	aAMSNetID	AT %I* 	:	AMSNETID;
	wSlaveADDR	AT %I*			:	WORD;
	PLCResetRequired	:	BOOL := FALSE;		
END_VAR

VAR_INPUT
	b_EnablePower 			: BOOL;
	r_CoolantTemperature 	: REAL;
END_VAR

VAR_OUTPUT
	Get : ST_HeatpumpSystemGet;
END_VAR

VAR
	PrimaryHeatpump_EnablePower		AT %Q* :	BOOL;
	SecondaryHeatpump_EnablePower	AT %Q* :	BOOL;
	b_AuxilliaryHeaterEnable		AT %Q*	:	Bool;
END_VAR

UpdateRTUSettings();				

CASE st_params.HeatpumpType OF
	eSupportedHeatpumps.TranePicco:
		PrimaryHeatpump := TraneHeatpump[0];
		TraneHeatpump[0](MBMaster := MBMaster, 
			ACPowerStatus := b_EnablePower,  
			st_params := st_params, 
			HeatPumpId := st_Params.PrimaryHeatpumpAddr);
		get.PrimaryHeatpumpGet REF= TraneHeatpump[0].Get;
				
	eSupportedHeatpumps.LgThermaV:
		PrimaryHeatpump := LGHeatpump[0];
		LGHeatpump[0](MBMaster := MBMaster, 
			ACPowerStatus := b_EnablePower,  
			st_params := st_params, 
			HeatPumpId := st_Params.PrimaryHeatpumpAddr);
		get.PrimaryHeatpumpGet REF= lgHeatpump[0].Get;
END_CASE

get.SecondaryHeatpumpGet REF= lgHeatpump[1].Get;

IF ST_Params.b_DoubleHeatpump THEN
	CASE st_params.HeatpumpType OF
		eSupportedHeatpumps.TranePicco:		
			SecondaryHeatpump := TraneHeatpump[1];
			TraneHeatpump[1](MBMaster := MBMaster, 
				ACPowerStatus := b_EnablePower,  
				st_params := st_params, 
				HeatPumpId := st_Params.SecondaryHeatpumpAddr,
				get => get.SecondaryHeatpumpGet);
		eSupportedHeatpumps.LgThermaV:		
			SecondaryHeatpump := LGHeatpump[1];	
			LGHeatpump[1](MBMaster := MBMaster, 
				ACPowerStatus := b_EnablePower,  
				st_params := st_params, 
				HeatPumpId := st_Params.SecondaryHeatpumpAddr,
				get => get.SecondaryHeatpumpGet);
	END_CASE
END_IF

get.HeatPumpStatus := get.PrimaryHeatpumpGet.HeatPumpState;
get.PrimaryHeatpumpGet.HeatpumpData.r_CoolantPower := CalculateCoolantPower();

PowerControl();
setMBControl();

METHOD CalculateCoolantPower : REAL
VAR_INST
	PowerMA : fb_MovingAverage := (enable := TRUE);
	ActualPower : REAL;
	
	deltaT :  REAL;
	cp	: REAL;
	Flow : REAL;
	
	ton_synctimer	: TON := (PT:= T#1S);
END_VAR
flow	:= get.PrimaryHeatpumpGet.HeatpumpData.ui_WaterFlowRate;
deltaT	:= get.PrimaryHeatpumpGet.HeatpumpData.r_InletWaterTemp - get.PrimaryHeatpumpGet.HeatpumpData.r_OutletWaterTemp;
cp		:= 3.647;

ton_synctimer(IN := NOT ton_synctimer.Q);

ActualPower := (flow * cp * deltaT * 1.05) / 0.06;

IF ton_synctimer.Q THEN
	PowerMA(IN := ActualPower, length:= 15);
END_IF

CalculateCoolantPower := PowerMA.Q;
END_METHOD

METHOD EMStop : BOOL
VAR_INPUT
END_VAR
EMstop := PrimaryHeatpump.emstop() and SecondaryHeatpump.emstop();
END_METHOD

METHOD GetDiagnostics 
VAR_IN_OUT
	AddError		: ARRAY [*] OF FB_AddErrorST;
	a_ActiveEvents	: ARRAY [*] OF ST_ErrorStruct;
	w_Index			: WORD;
END_VAR

VAR_OUTPUT
	b_errorActive	: BOOL;
	b_warningActive	: BOOL;
END_VAR

VAR
	by_errCt	: BYTE;
	by_warnCt	: BYTE;
	w_ID		: WORD;
END_VAR
(*Heatpump Heating inhibited*)	AddError[w_Index](
			b_ErrorTrig				:= b_AuxilliaryHeaterEnable,
			out_ST_Error			:= a_ActiveEvents[w_Index],
			w_ErrorID				:= 20,
			s_Message				:= 'Coolant undertemperature error, heatpump heating inhibited',
			e_sev					:= eSeverity.Info,	
			b_AutoClear				:= TRUE,
			);
		w_Index := w_Index +1;	
		
(*Heatpump type changed*)	AddError[w_Index](
			b_ErrorTrig				:= PLCResetRequired,
			out_ST_Error			:= a_ActiveEvents[w_Index],
			w_ErrorID				:= 21,
			s_Message				:= 'Heatpump type changed, Reset PLC to activate new settings',
			e_sev					:= eSeverity.Warning,	
			b_AutoClear				:= TRUE,
			);
		w_Index := w_Index +1;	

(*Heatpump type changed*)	AddError[w_Index](
			b_ErrorTrig				:= PLCResetRequired,
			out_ST_Error			:= a_ActiveEvents[w_Index],
			w_ErrorID				:= 22,
			s_Message				:= 'Heatpump not operational until PLC has been restarted!',
			e_sev					:= eSeverity.Warning,	
			b_AutoClear				:= TRUE,
			);
		w_Index := w_Index +1;	

//check if this call works:
PrimaryHeatpump.GetDiagnostics(AddError := AddError, a_ActiveEvents := a_ActiveEvents, w_Index := w_Index, b_errorActive => b_errorActive, b_warningActive => b_warningActive);
SecondaryHeatpump.GetDiagnostics(AddError := AddError, a_ActiveEvents := a_ActiveEvents, w_Index := w_Index, b_errorActive => b_errorActive, b_warningActive => b_warningActive);
END_METHOD

METHOD GetWearCounters : BOOL
VAR_INST
	MstrPowerCycles				:	FB_Varlogger;
	MstrPowerHours				:	FB_Varlogger;
	
	MstrCompressorCycles		:	FB_Varlogger;
	MstrWaterpumpHours			:	FB_Varlogger;
	
	SlowDataTimer				:	TON := (PT := T#1H);
END_VAR
SlowDataTimer(IN := NOT SlowDataTimer.Q);

MstrPowerCycles(		TriggerInput := PrimaryHeatpump_EnablePower,
						LogItemGroup := eLogItemGroupID.CoolingSystem, 
						LogItemName := 'MstrHPPwrCnt', 
						LogType := eLogtypes.TrackCycles);
						
MstrPowerCycles(		TriggerInput := PrimaryHeatpump_EnablePower,
						LogItemGroup := eLogItemGroupID.CoolingSystem, 
						LogItemName := 'MstrHPPwrHrs', 
						LogType := eLogtypes.TrackOnTime);

IF get.PrimaryHeatpumpGet.HeatpumpData.i_OperatingHours > 0 THEN
	Wearlogging.SetInteger(eLogItemGroupID.CoolingSystem, 	'MstrHPCompHrs', 			eLogTypes.WriteValue, 		INT_TO_LINT(get.PrimaryHeatpumpGet.HeatpumpData.i_OperatingHours));
END_IF

MstrCompressorCycles(	TriggerInput := ((get.PrimaryHeatpumpGet.HeatpumpData.r_HighPressure-get.PrimaryHeatpumpGet.HeatpumpData.r_LowPressure)>5), //test this
						LogItemGroup :=  eLogItemGroupID.CoolingSystem, 
						LogItemName := 'MstrHPCompCnt', 
						LogType := eLogtypes.TrackCycles);
END_METHOD

METHOD PRIVATE PowerControl : BOOL
VAR_INST
	PowerOnDelay1: TON := (PT := TIME#1S);
	PowerOnDelay2: TON := (PT := TIME#2S);
END_VAR

//heatpump 2 is enabled with a delay to limit inrush
PowerOnDelay1(in:= b_EnablePower, Q=>PrimaryHeatpump_EnablePower);
PowerOnDelay2(IN := b_EnablePower AND st_params.b_DoubleHeatpump ,Q=> SecondaryHeatpump_EnablePower);
END_METHOD

METHOD Reset : BOOL
VAR_INPUT
END_VAR
Reset := PrimaryHeatpump.Reset() and SecondaryHeatpump.Reset();
END_METHOD

METHOD PRIVATE SetMBControl : BOOL
VAR_INST
	ton_MaximumMBTimeframe	:	TON := (PT := TIME#10S);

	CommFreeForID			: BYTE := 0;
	CommFreeTimeout			: TON := (PT := TIME#10S);	
END_VAR
//500ms trigger to switch MB bus ownership to next heatpump
ton_MaximumMBTimeframe(in := NOT ton_MaximumMBTimeframe.Q);

IF NOT PrimaryHeatpump.MBCommBusy() AND NOT SecondaryHeatpump.MBCommBusy() THEN
	CommFreeForID := (CommFreeForID+1);
END_IF
	
PrimaryHeatPump.AllowMBComm(b_AllowComm := (CommFreeForID=1));
SecondaryHeatPump.AllowMBComm(b_AllowComm := (CommFreeForID=2));

IF CommFreeForID > SEL(st_params.b_DoubleHeatpump, 1, 2) THEN
	CommFreeForID := 0;
END_IF
END_METHOD

METHOD Shutdown : BOOL
VAR_INPUT
END_VAR
HeatPumpOperationAllowed := FALSE;
END_METHOD

METHOD Start : BOOL
VAR_INPUT
END_VAR
HeatpumpOperationAllowed := true;
END_METHOD

METHOD UpdateRTUSettings : BOOL
VAR_INPUT
END_VAR

VAR_INST
	CurrentBussettings			:	WORD 	:=  0;
	MethodSTate					:	UINT	:=	0;
	CoEWrite					:	FB_EcCoeSdoWriteEx;
	CoERead						:	FB_EcCoeSdoReadEx;
	Netid						:	T_AMSNETID;
	
	Testoutput					:	UDINT;
	Testbool					:	BOOL;
	TestBool2					:	BOOL;
	CurrentBusSetting			:   WORD;	
	RequiredBusSetting			:	WORD;	
	COEReadDone					:	F_trig;
	COEWriteDone				:	F_trig;
END_VAR
Netid := F_CreateAmsNetId(aAMSNetID);

CoERead(sNetID := Netid,
		nSlaveAddr := wSlaveADDR,
		nSubIndex := 0,
		nIndex := 16#4074,
		pDstBuf := ADR(CurrentBusSetting),
		cbBufLen := SIZEOF(CurrentBusSetting),
		tTimeout := T#1S,
		bCompleteAccess := TRUE,
		cbRead => Testoutput);

CoEWrite(sNetID := Netid,
		nSlaveAddr := wSlaveADDR,
		nSubIndex := 0,
		nIndex := 16#4074,
		pSRCBuf := ADR(RequiredBusSetting),
		cbBufLen := SIZEOF(RequiredBusSetting),
		tTimeout := T#1S,
		bCompleteAccess := TRUE);

COEReadDone(clk:= CoERead.bBusy);
COEwriteDone(clk:= CoEWrite.bBusy);


CASE MethodSTate OF
	0:	//init
		CoERead(bExecute := FALSE);
		CoEwrite(bExecute := FALSE);
		MethodSTate := 1;
	1:	//ReadCurrentSettings
		CoERead(bExecute := TRUE);
		IF COEReadDone.q THEN
			IF NOT CoERead.bError THEN
				MethodSTate := 2;
			END_IF
			CoERead(bExecute := FALSE);
		END_IF
	2:	//idle
		IF (st_params.HeatpumpType = eSupportedHeatpumps.LgThermaV AND CurrentBusSetting <> 3) THEN
			RequiredBusSetting := 3;
			MethodSTate := 3; //write new settings
		ELSIF(st_params.HeatpumpType = eSupportedHeatpumps.TranePicco AND CurrentBusSetting <> 4) THEN
			RequiredBusSetting := 4;			
			MethodSTate := 3; //write new settings
		END_IF
	3: //write new settings
		CoEwrite(bExecute := TRUE);
		IF COEWriteDone.q THEN
			CoEwrite(bExecute := False);
			IF NOT CoERead.bError THEN
				MethodSTate := 4;
			END_IF
			CoERead(bExecute := FALSE);
		END_IF
	4:	//Wait for reboot to activate settings
			PLCResetRequired := TRUE;
		
END_CASE
END_METHOD

METHOD WriteSetpoint : BOOL
VAR_INPUT
	OperatingMode	:	eHeatpumpMode := eHeatpumpMode.Standby;
	SetPoint		: 	REAL := 18.0;
END_VAR
IF HeatpumpOperationAllowed THEN
	IF Operatingmode = eHeatpumpMode.Heating AND r_CoolantTemperature < st_params.r_MinimumCoolantTemperatureForHPHeatingMode THEN
		PrimaryHeatpump.Setpoint(eHeatpumpMode.Standby, Temperature := 18.0);
		b_AuxilliaryHeaterEnable := TRUE;
	ELSE
		PrimaryHeatpump.Setpoint(OperatingMode := OperatingMode, Temperature:=SetPoint);
		b_AuxilliaryHeaterEnable := FALSE;
	END_IF
ELSE
	PrimaryHeatpump.Setpoint(eHeatpumpMode.Standby, Temperature := 18.0);
	b_AuxilliaryHeaterEnable := FALSE;
END_IF
//This method will also contain potential master/slave temperature differentials and other differences between heatpumps
//Heatpumps[2].WriteSetpoint(OperatingMode := OperatingMode);
END_METHOD

END_FUNCTION_BLOCK

// ---- POUs/Objects/CoolingSystem/HeatpumpSystem/FB_LGHeatpump.TcPOU
FUNCTION_BLOCK FB_LGHeatpump implements IF_Heatpump
VAR_IN_OUT
	MBMaster		:	ModbusRtuMasterV2_KL6x22B;
END_VAR

VAR_OUTPUT
	Get				:	ST_HeatPump_Get;

END_VAR

VAR_IN_OUT CONSTANT
	st_params		: 	ST_Coolingsystem_params;
END_VAR

VAR_INPUT
	ACPowerStatus	:	BOOL;
	HeatPumpID		:	BYTE;
	SFCInit			:	BOOL;
	e_ID				:	eObject_ID := eObject_ID.HeatPump;
END_VAR
		
VAR
	ton_MBBUSYTimeOut		: TON := (PT := T#10s);
	DataBuffer				:	ARRAY[0..50] OF WORD;
	ton_modbusStuckTrigger	:	Ton	:=	(PT := T#5S);
	Ton_ErrorTimer			:	Ton := (PT := T#5M);
	MBRetryCount			:	BYTE;
	MBFree					:	BOOL;
	bMBActive				:	BOOL;
	ftrig_ModbusStartTrigger		:	f_Trig;
	TransmissionDoneTrigger	:	F_Trig;
	rtrig_ManualModbusStartTrigger : r_trig;
	btest	:	BOOL;
	ManADDR : BYTE;
	ton_testTimer	:	Ton := (Pt := T#100MS);
	TP_ModbusStartTriggerDelay	:	TP := (PT := TIME#50MS);
	u_counter				:	UINT;
END_VAR

VAR
	RequestedSetpoint				:	st_OperatingPoint;
	b_EMStop						:	BOOL;
	b_resetErrors					:	BOOL;
	t_RemainingPreheatingTime	:	TIME;
	sPressureErrorText			:	STRING;
	sCompressorErrorText		:	STRING;
	sPumpErrorText				:	STRING;
	sWaterTempErrorText			:	STRING;
END_VAR

VAR PERSISTENT
	dt_LastHPOperationTime	:	DT := DT#1970-1-1-0:0:0.000;
END_VAR


VAR
	CoilStatus		:	BYTE;
	LGget	:	LG_get;
	LGset	:	LG_SET;

	HeatpumpEMOperationAvailable	:	Bool;
END_VAR

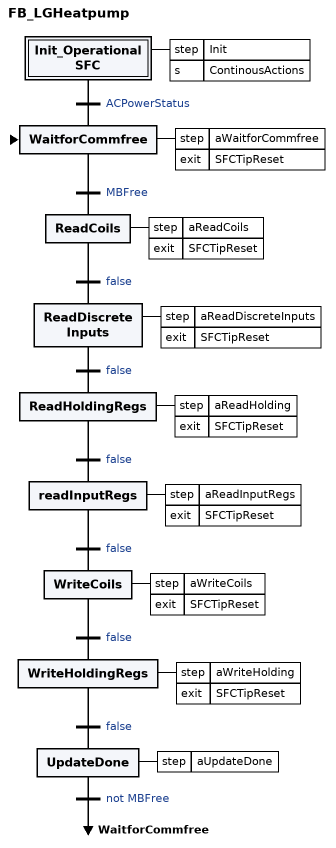
INITIAL_STEP Init_OperationalSFC:
    Init(N);  // step action
    ContinousActions(s);
END_STEP
TRANSITION FROM Init_OperationalSFC TO WaitforCommfree
    := ACPowerStatus;
END_TRANSITION
STEP WaitforCommfree:
    aWaitforCommfree(N);  // step action
    SFCTipReset(P0);  // exit action
END_STEP
TRANSITION FROM WaitforCommfree TO ReadCoils
    := MBFree;
END_TRANSITION
STEP ReadCoils:  // max time T#2S
    aReadCoils(N);  // step action
    SFCTipReset(P0);  // exit action
END_STEP
TRANSITION FROM ReadCoils TO ReadDiscreteInputs
    := false;
END_TRANSITION
STEP ReadDiscreteInputs:
    aReadDiscreteInputs(N);  // step action
    SFCTipReset(P0);  // exit action
END_STEP
TRANSITION FROM ReadDiscreteInputs TO ReadHoldingRegs
    := false;
END_TRANSITION
STEP ReadHoldingRegs:
    aReadHolding(N);  // step action
    SFCTipReset(P0);  // exit action
END_STEP
TRANSITION FROM ReadHoldingRegs TO readInputRegs
    := false;
END_TRANSITION
STEP readInputRegs:
    aReadInputRegs(N);  // step action
    SFCTipReset(P0);  // exit action
END_STEP
TRANSITION FROM readInputRegs TO WriteCoils
    := false;
END_TRANSITION
STEP WriteCoils:
    aWriteCoils(N);  // step action
    SFCTipReset(P0);  // exit action
END_STEP
TRANSITION FROM WriteCoils TO WriteHoldingRegs
    := false;
END_TRANSITION
STEP WriteHoldingRegs:
    aWriteHolding(N);  // step action
    SFCTipReset(P0);  // exit action
END_STEP
TRANSITION FROM WriteHoldingRegs TO UpdateDone
    := false;
END_TRANSITION
STEP UpdateDone:
    aUpdateDone(N);  // step action
END_STEP
TRANSITION FROM UpdateDone TO WaitforCommfree
    := not MBFree;
END_TRANSITION

METHOD AllowMBComm : BOOL
VAR_INPUT
	b_AllowComm	:	Bool;
END_VAR
MBFree	:= b_AllowComm;
END_METHOD

ACTION aReadCoils:
bMBActive := TRUE;

MBMaster.ReadCoils(	UnitID 		:= 	HeatPumpID,
					Quantity 	:= 	5,
					MBAddr		:=	0,				
					cbLength 	:= 	6,
					pMemoryAddr	:=	ADR(CoilStatus),
					Execute		:=	ftrig_ModbusStartTrigger.Q,
				);
	

IF TransmissionDoneTrigger.q THEN
	IF NOT MBMaster.Error THEN
		//Full datastruct for debug purposes. Can be removed later
		LGget.Coils.b_EnableOperation := CoilStatus.0;
		LGget.Coils.b_EnableSwwOperation := CoilStatus.1;
		LGget.Coils.b_EnableSilentMode := CoilStatus.2;
		LGget.Coils.b_EnableDesinfectionMode := Coilstatus.3;
		LGget.Coils.b_EmstopActive := CoilStatus.4;
		LGget.Coils.b_EnableEmStop := CoilStatus.5;
		//Full datastruct for debug purposes. Can be removed later
		
	ELSE
		MBRetryCount := MBRetryCount + 1;
	END_IF
	
	sfctip := TRUE;
END_IF


get.HeatpumpData.w_ErrorList[1] := lgget.Data.UI_ErrorCode;
get.Setpoint := lgget.Control.r_Setpoint1;
END_ACTION

ACTION aReadDiscreteInputs:


MBMaster.ReadInputStatus(	UnitID 		:= 	HeatPumpID,
							Quantity 	:= 	16,
							MBAddr		:=	0,
							cbLength 	:= 	SIZEOF(Databuffer),
							pMemoryAddr	:=	ADR(DataBuffer),
							Execute		:=	ftrig_ModbusStartTrigger.Q,
						);



IF TransmissionDoneTrigger.q THEN
	IF NOT MBMaster.Error THEN
		//Full datastruct for debug purposes. Can be removed later
		LGget.Status.b_WaterFlowNOK := DataBuffer[0].0;
		LGget.Status.b_WaterPumpOn := DataBuffer[0].1;
		LGget.Status.b_ExtWaterPumpOn := DataBuffer[0].2;
		LGget.Status.b_CompressorOn := DataBuffer[0].3;
		LGget.Status.b_DefrostOn := DataBuffer[0].4;
		LGget.Status.b_SWWModeOn := DataBuffer[0].5;
		LGget.Status.b_SWWTankDesinfectionActive := DataBuffer[0].6;
		LGget.Status.b_SilentModeOn := DataBuffer[0].7;
		LGget.Status.b_CoolingActive := DataBuffer[0].8;
		LGget.Status.b_SolarPumpActive := DataBuffer[0].9;
		LGget.Status.b_BackupHeater1Active := DataBuffer[0].10;
		LGget.Status.b_BackupHeater2Active := DataBuffer[0].11;
		LGget.Status.b_SWWBoostHeaterActive := DataBuffer[0].12;
		LGget.Status.b_ErrorActive := DataBuffer[0].13;
		LGget.Status.b_EMOperationAvailable := DataBuffer[0].14;
		LGget.Status.b_EMSWWOperationAvailable := DataBuffer[0].15;
		LGget.Status.b_MixPumpActive := DataBuffer[1].0;
		//Full datastruct for debug purposes. Can be removed later
		
		get.Events.b_PumpError := DataBuffer[0].0;
		get.HeatpumpData.b_DefrostingActive := DataBuffer[0].4;
		
		
		//error active and no em operation allowed
		IF DataBuffer[0].13 THEN
			get.HeatPumpState := eHeatpumpstate.ERROR;
			IF NOT DataBuffer[0].14 THEN
				HeatpumpEMOperationAvailable := FALSE;
			ELSE
				HeatpumpEMOperationAvailable := TRUE;
			END_IF
		ELSIF get.HeatPumpState = eHeatpumpstate.ERROR THEN
			get.HeatPumpState := eHeatpumpstate.Initializing;
			HeatpumpEMOperationAvailable := FALSE;
		END_IF
		
		//done, preset for next step
		MBRetryCount := 0;
	ELSE
		MBRetryCount := MBRetryCount + 1;
	END_IF
	sfctip := TRUE;
END_IF
END_ACTION

ACTION aReadHolding:

MBMaster.ReadRegs(	UnitID 		:= 	HeatPumpID,
					Quantity 	:= 	10,
					MBAddr		:=	0,
					cbLength 	:= 	SIZEOF(Databuffer),
					pMemoryAddr	:=	ADR(DataBuffer),
					Execute		:=	ftrig_ModbusStartTrigger.Q,
					);


IF TransmissionDoneTrigger.q THEN
	IF NOT MBMaster.Error THEN
		LGget.Control.ui_OperatingMode := Databuffer[0];
		LGget.Control.ui_ControlMode := Databuffer[1];
		LGget.Control.r_Setpoint1 := (WORD_TO_REAL(Databuffer[2])/10);
		LGget.Control.r_RoomSetpoint := (WORD_TO_REAL(Databuffer[3])/10);
		LGget.Control.ui_TempShiftValue := Databuffer[4];
		LGget.Control.r_Setpoint2 := (WORD_TO_REAL(Databuffer[5])/10);
		LGget.Control.r_RoomSetpoint2 := (WORD_TO_REAL(Databuffer[6])/10);
		LGget.Control.ui_TempShiftValue2 := Databuffer[7];
		LGget.Control.r_DHWgoalTemp := (WORD_TO_REAL(Databuffer[8])/10);
		LGget.Control.ui_EnergyStatus := Databuffer[9];
		
		get.Setpoint := (WORD_TO_REAL(Databuffer[2])/10);


		IF get.HeatPumpState <> eHeatpumpstate.ERROR THEN
			CASE lgget.Data.ui_OperationalMode OF
				0:
					get.HeatPumpState := eHeatpumpstate.Standby;
				1:
					get.HeatPumpState := eHeatpumpstate.Active_Cooling;
				2:
					get.HeatPumpState := eHeatpumpstate.Active_Heating;
			END_CASE
		END_IF
	
		//done, preset for next step
		MBRetryCount := 0;

	ELSE
		MBRetryCount := MBRetryCount + 1;
		
	END_IF
	sfctip := TRUE;
END_IF
END_ACTION

ACTION aReadInputRegs:
//SFCTip := FALSE;

MBMaster.ReadInputRegs ( 
					UnitID 		:= 	HeatPumpID,
					Quantity 	:= 	13,
					MBAddr		:=	0,
					cbLength 	:= 	SIZEOF(Databuffer),
					pMemoryAddr	:=	ADR(Databuffer),
					Execute		:=	ftrig_ModbusStartTrigger.Q,		
					);
				
IF TransmissionDoneTrigger.q THEN
	IF NOT MBMaster.Error THEN
		
	//Full datastruct for debug purposes. Can be removed later
		LGget.Data.UI_ErrorCode := Databuffer[0];	
		LGget.Data.ui_OperationalMode := (Databuffer[1]);	
		LGget.Data.r_CoolantInletTemp := WORD_TO_REAL((Databuffer[2]))/10;	
		LGget.Data.r_CoolantOutletTemp := WORD_TO_REAL((Databuffer[3]))/10;
		LGget.Data.r_BackupHeaterTemp := WORD_TO_REAL((Databuffer[4]))/10;
		LGget.Data.r_SWWTankTemp :=  WORD_TO_REAL((Databuffer[5]))/10;
		LGget.Data.r_SolarCollectorTemp := WORD_TO_REAL((Databuffer[6]))/10;
		LGget.Data.r_RoomTemp1 := WORD_TO_REAL((Databuffer[7]))/10;
		LGget.Data.r_FlowRate := WORD_TO_REAL((Databuffer[8]))/10;
		LGget.Data.r_FlowTempCircuit2 := WORD_TO_REAL((Databuffer[9]))/10;
		LGget.Data.r_RoomTemp2 := WORD_TO_REAL((Databuffer[10]))/10;
		LGget.Data.UI_EnergyStatus := (Databuffer[11]);
		LGget.Data.r_OutsideTemp := WORD_TO_REAL((Databuffer[12]))/10;
	//full datastruct for debug purposes. can be removed later	
		
		
		get.HeatpumpData.w_ErrorList[1] := Databuffer[0];
		Get.HeatpumpData.r_InletWaterTemp := WORD_TO_REAL((Databuffer[2]))/10;	
		get.HeatpumpData.r_OutletWaterTemp := WORD_TO_REAL((Databuffer[3]))/10;
		get.HeatpumpData.r_OutdoorTemp := WORD_TO_REAL((Databuffer[12]))/10;
		get.HeatpumpData.ui_WaterFlowRate := TO_UINT(Databuffer[8]/10);
	ELSE
		MBRetryCount := MBRetryCount + 1;
	END_IF
	sfctip := TRUE;
END_IF
END_ACTION

ACTION aUpdateDone:
SFCTip := FALSE;
bMBActive := FALSE;
END_ACTION

ACTION aWaitforCommfree:
//SFCTip := FALSE;
//b_EnableTransmission	:= FALSE;
//ModbusStartTrigger(clk := b_EnableTransmission);
END_ACTION

ACTION aWriteCoils:


CoilStatus.0 := requestedSetpoint.OperatingMode <> eHeatpumpMode.Standby; // operation off

CoilStatus.5 := EMHeatingModeRequired();


//IF get.HeatPumpState = eHeatpumpState.Initializing THEN
	MBMaster.WriteMultipleCoils(	UnitID 		:= 	HeatPumpID,
									Quantity 	:= 	5,
									MBAddr		:=	0,
									cbLength 	:= 	1,
									pMemoryAddr	:=	ADR(CoilStatus),
									Execute		:=	ftrig_ModbusStartTrigger.Q,	
						);
	
	IF TransmissionDoneTrigger.q THEN
		IF NOT MBMaster.Error THEN
			sfctip := TRUE;
			
		ELSE
			MBRetryCount := MBRetryCount + 1;
			sfctip := NOT sfctip;
		END_IF
	END_IF
//ELSE
//	sfctip := NOT sfctip;
//END_IF
END_ACTION

ACTION aWriteHolding:

CASE requestedSetpoint.OperatingMode OF
	eHeatpumpMode.Cooling:
		Databuffer[0] := 0; // cooling mode
		Databuffer[2] := REAL_TO_WORD(requestedSetpoint.Setpoint*10);
	eHeatpumpMode.Heating:
		Databuffer[0] := 4; // Heating mode
		Databuffer[2] := REAL_TO_WORD(requestedSetpoint.Setpoint*10);	
END_CASE
		
Databuffer[1] := 1; // inlet temperature control
Databuffer[3] := 0;
Databuffer[4] := 0;
Databuffer[5] := 0;
Databuffer[6] := 0;
Databuffer[7] := 0;
Databuffer[8] := 0;
Databuffer[9] := 2; // normal operation

MBMaster.WriteRegs (
		UnitID 		:= 	HeatPumpID,
		Quantity 	:= 	10,
		MBAddr		:=	0,
		cbLength 	:= 	SIZEOF(Databuffer),
		pMemoryAddr	:=	ADR(Databuffer),
		Execute		:=	ftrig_ModbusStartTrigger.Q,		
);



IF TransmissionDoneTrigger.q THEN
	IF NOT MBMaster.Error THEN
		//done, preset for next step

		MBRetryCount := 0;;
	ELSE
		MBRetryCount := MBRetryCount + 1;
	END_IF
	sfctip := TRUE;
END_IF
END_ACTION

ACTION ContinousActions:
//sfctip := False;
ton_modbusStuckTrigger(in := NOT ton_modbusStuckTrigger.q AND NOT TP_ModbusStartTriggerDelay.q);
TP_ModbusStartTriggerDelay(IN := NOT MBMaster.BUSY AND NOT ton_modbusStuckTrigger.q );
ftrig_ModbusStartTrigger(clk := TP_ModbusStartTriggerDelay.Q);

IF SFCError THEN
	SFCError := FALSE;
	get.Events.b_CommWarning := TRUE;
END_IF

IF NOT ACPowerStatus THEN
	IF get.HeatPumpState <> eHeatpumpstate.OFF THEN
		SFCReset := TRUE;
	END_IF
ELSIF get.HeatPumpState = eHeatpumpState.OFF THEN
	get.HeatPumpState := eHeatpumpState.Initializing;
END_IF

//safeguard, should the sfc get stuck, heatpumpsystem can revoke MB rights and SFC resets.
//IF NOT MBfree AND bMBActive AND NOT MBMaster.BUSY THEN
//	SFCReset := TRUE;
//END_IF 



HeatpumpPreheatControl();


//reset mb master if stuck in busy
ton_MBBUSYTimeOut(IN := MBmaster.BUSY);
IF ton_MBBUSYTimeOut.Q THEN
	MBMaster.ReadCoils();
	MBMaster.ReadInputStatus();
	MBMaster.ReadRegs();
	MBMaster.WriteMultipleCoils();
	MBMaster.WriteRegs();
	MBMaster.WriteSingleRegister();
END_IF

//Reset heatpump when error occurs, but after a bit of cooldown time.
//Maybe add a functionality to stop trying after x tries to prevent continuous reset cycles
Ton_ErrorTimer(in := get.Events.b_CompressorError OR 
					get.Events.b_FanError OR 
					get.Events.b_PressureError OR 
					get.Events.b_WaterTempError OR 
					get.Events.b_PumpError );
IF Ton_ErrorTimer.Q THEN
	b_resetErrors := TRUE;
END_IF

TransmissionDoneTrigger(clk := MBMaster.Busy);
MBMaster.Timeout		:= st_params.t_ModbusTimeOut;		

get.Events.b_CommWarning := MBRetryCount > st_params.i_modbusRetries;

IF TRUE THEN
	CASE requestedSetpoint.OperatingMode OF
		eHeatPumpMode.Standby:
			LGset.Coils.b_EnableOperation := FALSE;
			LGset.Regs.ui_OperatingMode := 3;
		eHeatPumpMode.Cooling:
			LGset.Coils.b_EnableOperation := TRUE;
			LGset.Regs.r_Setpoint1 := RequestedSetpoint.Setpoint;
			LGset.Regs.ui_OperatingMode := 0;
		eHeatPumpMode.Heating:
			LGset.Coils.b_EnableOperation := TRUE;
			LGset.Regs.r_Setpoint1 := RequestedSetpoint.Setpoint;
			LGset.Regs.ui_OperatingMode := 4;
	END_CASE
END_IF
END_ACTION

METHOD EMHeatingModeRequired : BOOL
VAR_INPUT
END_VAR
//some heatpump faults allow for emergency heating operation. If this occurs and heating is required, switch to emergency heating mode to keep the system warm.
//Cooling operation is not available in this mode.

IF lgget.Status.b_EMOperationAvailable AND RequestedSetpoint.OperatingMode = eHeatpumpmode.Heating THEN
	EMHeatingModeRequired := TRUE;
ELSE
	EMHeatingModeRequired := FALSE;
END_IF
END_METHOD

METHOD EMStop : BOOL
RequestedSetpoint.OperatingMode := eHeatpumpMode.Standby;
b_Emstop := TRUE;
EMstop := TRUE;
END_METHOD

METHOD GetDiagnostics 
VAR_IN_OUT
	AddError		: ARRAY [*] OF FB_AddErrorST;
	a_ActiveEvents	: ARRAY [*] OF ST_ErrorStruct;
	w_Index			: WORD;
END_VAR

VAR_OUTPUT
	b_errorActive	: BOOL;
	b_warningActive	: BOOL;
END_VAR

VAR
	by_errCt	: BYTE;
	by_warnCt	: BYTE;
	HPErrorText	: STRING;
END_VAR
	(*Modbus comm fault*)	AddError[w_Index](
			b_ErrorTrig			:= Get.Events.b_commwarning,
			out_ST_Error			:= a_ActiveEvents[w_Index],
			w_ErrorID				:= 30 + ((HeatPumpID-1)*10),
			e_ObjectID				:= e_ID,
			s_Message				:= 'Modbus communication fault',
			e_sev					:= eSeverity.Warning,	
			b_AutoClear			:= TRUE,
			t_TriggerTime		:=	T#60s,
			//in_e_ErrAckAccess		:= TRUE,
			);
		w_Index := w_Index +1;
		
CASE get.HeatpumpData.w_ErrorList[1] OF
	0:										HPErrorText := '';
	1, 8, 13, 19, 44:						HPErrorText := 'Misc Sensor error';
	2, 6, 16, 17, 18, 41, 45, 46, 65, 114:	HPErrorText := 'Temperature sensor error';
	10:										HPErrorText := 'Water pump blocked';
	3, 5, 53, 52:							HPErrorText := 'Internal comm error';
	9, 60:									HPErrorText := 'Eeprom error';
	14:										HPErrorText := 'Flow error';
	15:										HPErrorText := 'Water outlet overheat';
	20:										HPErrorText := 'Heater thermal fuse failed';
	21, 22, 27, 29:							HPErrorText := 'Compressor overcurrent';
	26: 									HPErrorText := 'Compressor fault';
	32: 									HPErrorText := 'Compressor output overtemperature';
	23: 									HPErrorText := 'DC Voltage error';
	35: 									HPErrorText := 'Low pressure error';
	43:   									HPErrorText := 'pressure sensor error';
	54:   									HPErrorText := 'Input phase error';
	61:   									HPErrorText := 'condensor overtemperature error';
	62:   									HPErrorText := 'heatsink overtemperature error'; 
	67:  									HPErrorText := 'Fan blocked error';
ELSE
	HPErrorText := 'Unknown error';
END_CASE


		
	(*Heatpump fault*)	AddError[w_Index](
			b_ErrorTrig				:= get.HeatpumpData.w_ErrorList[1] <> 0,
			out_ST_Error			:= a_ActiveEvents[w_Index],
			w_ErrorID				:= 31 + ((HeatPumpID-1)*10),
			s_Message				:= concat(concat(concat('Heatpump fault: ', TO_STRING(get.HeatpumpData.w_ErrorList[1])), ' :'), HPErrorText),
			e_sev					:= eSeverity.Warning,	
			b_AutoClear				:= True,
			t_TriggerTime			:=	T#1S,
			//in_e_ErrAckAccess		:= TRUE,
			);
		w_Index := w_Index +1;
	
	
	(*Heatpump warning*)			AddError[w_Index](
			b_ErrorTrig			:= LGGet.Coils.b_EnableSwwOperation AND lgget.Status.b_EMOperationAvailable,
			out_ST_Error		:= a_ActiveEvents[w_Index],
			w_ErrorID			:= 32 + ((HeatPumpID-1)*10),
			s_Message			:= 'Emergency operation active, performance may be restricted',
			e_sev				:= eSeverity.Warning,	
			b_AutoClear			:= FALSE,
			t_TriggerTime		:=	T#1S,
			//in_e_ErrAckAccess		:= TRUE,
			);
		w_Index := w_Index +1;
		

//	(*Heatpump Pump fault*)			AddError[w_Index](
//			b_ErrorTrig			:= Get.Events.b_PumpError,
//			out_ST_Error			:= a_ActiveEvents[w_Index],
//			w_ErrorID				:= 33 + ((HeatPumpID-1)*10),
//			s_Message				:= 'pump fault',
//			e_sev					:= eSeverity.Warning,	
//			b_AutoClear			:= FALSE,
//			t_TriggerTime		:=	T#1S,
//			//in_e_ErrAckAccess		:= TRUE,
//			);
//		w_Index := w_Index +1;	
		
	(*Heatpump Preheating active*)			AddError[w_Index](
			b_ErrorTrig				:= Get.Events.b_HeatpumpPreheatingActive,
			out_ST_Error			:= a_ActiveEvents[w_Index],
			w_ErrorID				:= 34 + ((HeatPumpID-1)*10),
			s_Message				:= concat('Heatpump preheating active for ', TO_STRING(t_RemainingPreheatingTime)),
			e_sev					:= eSeverity.Info,	
			b_AutoClear				:= TRUE,
			);
		w_Index := w_Index +1;
END_METHOD

METHOD PRIVATE HeatpumpPreheatControl : BOOL
VAR
	b_PreheatingRequired	:	BOOL;
END_VAR

VAR_INST
	ton_PreheatingTimer	:	Ton;
END_VAR
//enable operation
ton_PreheatingTimer(IN:= ACPowerStatus, PT:= TO_TIME(st_params.dw_HeatpumpOperationDelay*1000*60));
b_PreheatingRequired := ((DT_TO_INT(GVL.dt_SystemDateTime) - DT_TO_INT(dt_LastHPOperationTime))/60) > st_params.i_SkipHPPreheatingTime;

t_RemainingPreheatingTime := ton_PreheatingTimer.PT - ton_preheatingTimer.ET;

IF ton_PreheatingTimer.Q THEN
	dt_LastHPOperationTime := GVL.dt_SystemDateTime;
	t_RemainingPreheatingTime := T#0ms;
END_IF

get.Events.b_HeatpumpPreheatingActive := b_PreheatingRequired AND ACPowerStatus ;
END_METHOD

ACTION Init:
get.HeatPumpState := eHeatpumpstate.OFF;
bmbActive := FALSE;
SFCReset := FALSE;
get.Events.b_CommWarning := FALSE;
MBRetryCount := 0;
END_ACTION

METHOD MBCommBusy : BOOL
VAR_INPUT
END_VAR
MBCommBusy := bMBActive;
END_METHOD

METHOD ParseHeatPumpErrors : BOOL
VAR_INPUT
	w_Alarms1	:	WORD;
	w_Alarms2	:	WORD;
	w_Alarms3	:	WORD;
	w_Alarms4	:	WORD;
	w_Alarms5	:	WORD;
	w_Alarms6	:	WORD;
	w_Alarms7	:	WORD;
END_VAR		


VAR_IN_OUT
	get	:	ST_HeatPump_Get;	
END_VAR




get.events.b_ProbeError		:=	WORD_TO_BOOL(w_Alarms3) OR WORD_TO_BOOL(w_Alarms4) OR w_Alarms5.0;

get.events.b_PressureError		:=	w_Alarms1.0 OR	//E001: High Pressure
									w_Alarms1.1 OR //E002: Low Pressure
									w_Alarms2.3;	//E020: Inverted Pressure Transducers
									
sPressureErrorText := '';
IF get.events.b_PressureError THEN
	sPressureErrorText := concat(sPressureErrorText, SEL(w_Alarms1.0, '', ' E001'));
	sPressureErrorText := concat(sPressureErrorText, SEL(w_Alarms1.1, '', ' E002'));
	sPressureErrorText := concat(sPressureErrorText, SEL(w_Alarms2.3, '', ' E020'));
END_IF
									
get.events.b_CompressorError	:=	w_Alarms1.2 OR //E003: Compressor overheated
									w_Alarms1.7 OR //E008: Compressor underspeed
									w_Alarms1.8 OR	//E009: High disch temp
									w_Alarms1.12 OR //E013: Comp2 Overheated
									w_Alarms2.2 OR	//E019: CP2 High disch temp
									w_Alarms2.6 OR	//E023: Comp3 Overheated
									w_Alarms5.1 OR //'E801: Link Inverter1',
									w_Alarms5.2 OR //'E802: Link Inverter2',
									w_Alarms5.3 OR //'E803: Link Inverter3',
									w_Alarms5.4 OR //'E851: HWfault Inverter1',
									w_Alarms5.5 OR //'E852: HWfault Inverter2',
									w_Alarms5.6 OR //'E853: HWfault Inverter3',
									w_Alarms5.7 OR //'E861: OverCurrent Inv1',
									w_Alarms5.8 OR //'E862: OverCurrent Inv2',
									w_Alarms5.9 OR //'E863: OverCurrent Inv3',
									w_Alarms5.10 OR //'E871: High Temp Inv1',
									w_Alarms5.11 OR //'E872: High Temp Inv2',
									w_Alarms5.12 OR //'E873: High Temp Inv3',
									w_Alarms5.13 OR //'E881: Bad Voltage Inv1',
									w_Alarms5.14 OR //'E882: Bad Voltage Inv2',
									w_Alarms5.15 OR //'E883: Bad Voltage Inv3',
									w_Alarms6.0 OR //E891: Phase Seq Inv1',
									w_Alarms6.1 OR //'E892: Phase Seq Inv2',
									w_Alarms6.2 OR //'E893: Phase Seq Inv3',
									w_Alarms6.3 OR //'E901: Model err Inv1',
									w_Alarms6.4 OR //'E902: Model err Inv2',
									w_Alarms6.5 OR //'E903: Model err Inv3',
									w_Alarms6.6 OR //'E911: Ovl error Inv1',
									w_Alarms6.7 OR //'E9112: Ovl error Inv2',
									w_Alarms6.8 OR //'E913: Ovl error Inv3',
									w_Alarms6.9 OR //'E921: Overc PFC Inv1',
									w_Alarms6.10 OR //'E922: Overc PFC Inv2',
									w_Alarms6.11 OR //'E923: Overc PFC Inv3',
									w_Alarms6.12 OR //'E931: Int Com ERR Inv1',
									w_Alarms6.13 OR //'E932: Int Com ERR Inv2',
									w_Alarms6.14 OR //'E933: Int Com ERR Inv3',
									w_Alarms6.15 OR //'E941: Fault PFC Inv1',
									w_Alarms7.0 OR //E942: Fault PFC Inv2
									w_Alarms7.1 OR //'E943: Fault PFC Inv3',
									w_Alarms7.2 OR //'E951: Probe error Inv1',
									w_Alarms7.3 OR //'E952: Probe error Inv2',
									w_Alarms7.4 OR //'E953: Probe error Inv3',
									w_Alarms7.5 OR //'E961: Abnormal Cond Inv1',
									w_Alarms7.6 OR //'E962: Abnormal Cond Inv2',
									w_Alarms7.7 OR //'E963: Abnormal Cond Inv3',
									w_Alarms7.8 OR //'E971: Inv1 Eeprom Error',
									w_Alarms7.9 OR //'E972: Inv2 Eeprom Error',
									w_Alarms7.10 OR //'E973: Inv3 Eeprom Error',
									w_Alarms7.11;	//E029: CP3 High disch temp

sCompressorErrorText := '';
IF get.events.b_CompressorError THEN
	sCompressorErrorText := concat(sCompressorErrorText, SEL(w_Alarms1.2, '', ' E003'));
	sCompressorErrorText := concat(sCompressorErrorText, SEL(w_Alarms1.7, '', ' E008'));
	sCompressorErrorText := concat(sCompressorErrorText, SEL(w_Alarms1.8, '', ' E009'));
	sCompressorErrorText := concat(sCompressorErrorText, SEL(w_Alarms1.12, '', ' E013'));
	sCompressorErrorText := concat(sCompressorErrorText, SEL(w_Alarms2.2, '', ' E019'));
	sCompressorErrorText := concat(sCompressorErrorText, SEL(w_Alarms2.6, '', ' E023'));
	sCompressorErrorText := concat(sCompressorErrorText, SEL(w_Alarms5.1, '', ' E801'));
	sCompressorErrorText := concat(sCompressorErrorText, SEL(w_Alarms5.2, '', ' E802'));
	sCompressorErrorText := concat(sCompressorErrorText, SEL(w_Alarms5.3, '', ' E803'));
	sCompressorErrorText := concat(sCompressorErrorText, SEL(w_Alarms5.4, '', ' E851'));
	sCompressorErrorText := concat(sCompressorErrorText, SEL(w_Alarms5.5, '', ' E852'));
	sCompressorErrorText := concat(sCompressorErrorText, SEL(w_Alarms5.6, '', ' E853'));
	sCompressorErrorText := concat(sCompressorErrorText, SEL(w_Alarms5.7, '', ' E861'));
	sCompressorErrorText := concat(sCompressorErrorText, SEL(w_Alarms5.8, '', ' E862'));
	sCompressorErrorText := concat(sCompressorErrorText, SEL(w_Alarms5.9, '', ' E863'));
	sCompressorErrorText := concat(sCompressorErrorText, SEL(w_Alarms5.10, '', ' E871'));
	sCompressorErrorText := concat(sCompressorErrorText, SEL(w_Alarms5.11, '', ' E872'));
	sCompressorErrorText := concat(sCompressorErrorText, SEL(w_Alarms5.12, '', ' E873'));
	sCompressorErrorText := concat(sCompressorErrorText, SEL(w_Alarms5.13, '', ' E881'));
	sCompressorErrorText := concat(sCompressorErrorText, SEL(w_Alarms5.14, '', ' E882'));
	sCompressorErrorText := concat(sCompressorErrorText, SEL(w_Alarms5.15, '', ' E883'));
	sCompressorErrorText := concat(sCompressorErrorText, SEL(w_Alarms6.0 , '', ' E891'));
	sCompressorErrorText := concat(sCompressorErrorText, SEL(w_Alarms6.1 , '', ' E892'));
	sCompressorErrorText := concat(sCompressorErrorText, SEL(w_Alarms6.2 , '', ' E893'));
	sCompressorErrorText := concat(sCompressorErrorText, SEL(w_Alarms6.3 , '', ' E901'));
	sCompressorErrorText := concat(sCompressorErrorText, SEL(w_Alarms6.4 , '', ' E902'));
	sCompressorErrorText := concat(sCompressorErrorText, SEL(w_Alarms6.5 , '', ' E903'));
	sCompressorErrorText := concat(sCompressorErrorText, SEL(w_Alarms6.6 , '', ' E911'));
	sCompressorErrorText := concat(sCompressorErrorText, SEL(w_Alarms6.7 , '', ' E912'));
	sCompressorErrorText := concat(sCompressorErrorText, SEL(w_Alarms6.8 , '', ' E913'));
	sCompressorErrorText := concat(sCompressorErrorText, SEL(w_Alarms6.9 , '', ' E921'));
	sCompressorErrorText := concat(sCompressorErrorText, SEL(w_Alarms6.10, '', ' E922'));
	sCompressorErrorText := concat(sCompressorErrorText, SEL(w_Alarms6.11, '', ' E923'));
	sCompressorErrorText := concat(sCompressorErrorText, SEL(w_Alarms6.12, '', ' E931'));
	sCompressorErrorText := concat(sCompressorErrorText, SEL(w_Alarms6.13, '', ' E932'));
	sCompressorErrorText := concat(sCompressorErrorText, SEL(w_Alarms6.14, '', ' E933'));
	sCompressorErrorText := concat(sCompressorErrorText, SEL(w_Alarms6.15, '', ' E941'));
	sCompressorErrorText := concat(sCompressorErrorText, SEL(w_Alarms7.0 , '', ' E942'));
	sCompressorErrorText := concat(sCompressorErrorText, SEL(w_Alarms7.1 , '', ' E943'));
	sCompressorErrorText := concat(sCompressorErrorText, SEL(w_Alarms7.2 , '', ' E951'));
	sCompressorErrorText := concat(sCompressorErrorText, SEL(w_Alarms7.3 , '', ' E952'));
	sCompressorErrorText := concat(sCompressorErrorText, SEL(w_Alarms7.4 , '', ' E953'));
	sCompressorErrorText := concat(sCompressorErrorText, SEL(w_Alarms7.5 , '', ' E961'));
	sCompressorErrorText := concat(sCompressorErrorText, SEL(w_Alarms7.6 , '', ' E962'));
	sCompressorErrorText := concat(sCompressorErrorText, SEL(w_Alarms7.7 , '', ' E963'));
	sCompressorErrorText := concat(sCompressorErrorText, SEL(w_Alarms7.8 , '', ' E971'));
	sCompressorErrorText := concat(sCompressorErrorText, SEL(w_Alarms7.9 , '', ' E972'));
	sCompressorErrorText := concat(sCompressorErrorText, SEL(w_Alarms7.10, '', ' E973'));
	sCompressorErrorText := concat(sCompressorErrorText, SEL(w_Alarms7.11, '', ' E029'));
END_IF
								
get.events.b_ValveError		:=		w_Alarms2.11; //E041: Incongruent temps;


get.events.b_FanError			:=	w_Alarms1.2 OR //E004: Fan Overheated	
									w_Alarms1.13 OR //E014: Fan2 Overheated 
									w_Alarms2.7;	//E024: Fan3 Overheated					

get.events.b_PumpError			:=	w_Alarms1.5 OR	 	//E006: Lack of flow
									w_Alarms1.15 OR 	//E016: Pump Overheated
									w_Alarms2.9;		//E026: Pump2 Overheated

sPumpErrorText := '';
IF get.events.b_PumpError THEN
	sPumpErrorText := concat(sPumpErrorText, SEL(w_Alarms1.5, '', ' E006'));
	sPumpErrorText := concat(sPumpErrorText, SEL(w_Alarms1.15, '', ' E016'));
	sPumpErrorText := concat(sPumpErrorText, SEL(w_Alarms2.9, '', ' E026'));		
END_IF						
									
get.events.b_WaterTempError		:=	w_Alarms2.1 OR	//E018: OverTemperature
									w_Alarms1.4;	//E005: Frost

sWaterTempErrorText := '';									
IF get.events.b_WaterTempError THEN
	sWaterTempErrorText := concat(sWaterTempErrorText, SEL(w_Alarms1.5, '', ' E018'));
	sWaterTempErrorText := concat(sWaterTempErrorText, SEL(w_Alarms1.15, '', ' E005'));	
END_IF		


									
get.events.b_IOError			:=	w_Alarms2.14 OR 	//E101: IOMod1 Disconnected
									w_Alarms2.15; 		//E102: IOMod2 Disconnected
END_METHOD

METHOD Reset : BOOL
//until restarting the heatpump we don't know if errors are gone. So clear them for now.

get.Events.b_CompressorError := FALSE;
get.Events.b_FanError := FALSE;
get.Events.b_IOError := FALSE;
get.Events.b_PressureError := FALSE;
get.Events.b_ProbeError := FALSE;
get.Events.b_PumpError := FALSE;
get.Events.b_ValveError := FALSE;
get.Events.b_WaterTempError := FALSE;
get.Events.b_CommWarning := FALSE;
b_Emstop := FALSE;

MBRetryCount := 0;
Reset := true;
END_METHOD

METHOD Setpoint : BOOL
VAR_INPUT
	OperatingMode	:	eHeatpumpMode	:= 	eHeatpumpMode.Standby;
	Temperature		: 	REAL			:=	18;
END_VAR
IF get.HeatPumpState >= eHeatpumpstate.Standby AND 
	NOT get.Events.b_HeatpumpPreheatingActive AND 
	NOT b_EMstop THEN
	RequestedSetpoint.Setpoint		:= Temperature;
	RequestedSetpoint.OperatingMode := OperatingMode;
ELSE
	RequestedSetpoint.OperatingMode := eHeatPumpMode.Standby;
	RequestedSetpoint.Setpoint		:= 18.0;
END_IF

get.Setpoint := RequestedSetpoint.Setpoint;
END_METHOD

ACTION SFCTipReset:
SFCTip := FALSE;
END_ACTION

METHOD VariableMapping : BOOL
VAR_INPUT
END_VAR
END_METHOD

END_FUNCTION_BLOCK

// ---- POUs/Objects/CoolingSystem/HeatpumpSystem/FB_TraneHeatpump.TcPOU
FUNCTION_BLOCK FB_TraneHeatpump implements IF_Heatpump
VAR_IN_OUT
	MBMaster		:	ModbusRtuMasterV2_KL6x22B;
END_VAR

VAR_OUTPUT
	Get				:	ST_HeatPump_Get;

END_VAR

VAR_IN_OUT CONSTANT
	st_params		: 	ST_Coolingsystem_params;
END_VAR

VAR_INPUT
	ACPowerStatus	:	BOOL;
	HeatPumpID		:	BYTE;
	SFCInit			:	BOOL;
	e_ID				:	eObject_ID := eObject_ID.HeatPump;
END_VAR
		
VAR
	ton_MBBUSYTimeOut		: TON := (PT := T#10s);
	DataBuffer				:	ARRAY[0..50] OF WORD;
	ton_modbusStuckTrigger	:	Ton	:=	(PT := T#5S);
	Ton_ErrorTimer			:	Ton := (PT := T#5M);
	MBRetryCount			:	BYTE;
	MBFree					:	BOOL;
	bMBActive				:	BOOL;
	ftrig_ModbusStartTrigger		:	f_Trig;
	TransmissionDoneTrigger	:	F_Trig;
	
	TP_ModbusStartTriggerDelay	:	TP := (PT := TIME#50MS);
	u_counter				:	UINT;
END_VAR

VAR
	RequestedSetpoint				:	st_OperatingPoint;
	b_EMStop						:	BOOL;
	b_resetErrors					:	BOOL;
	t_RemainingPreheatingTime	:	TIME;
	sPressureErrorText			:	STRING;
	sCompressorErrorText		:	STRING;
	sPumpErrorText				:	STRING;
	sWaterTempErrorText			:	STRING;
END_VAR

VAR PERSISTENT
	dt_LastHPOperationTime	:	DT := DT#1970-1-1-0:0:0.000;
END_VAR

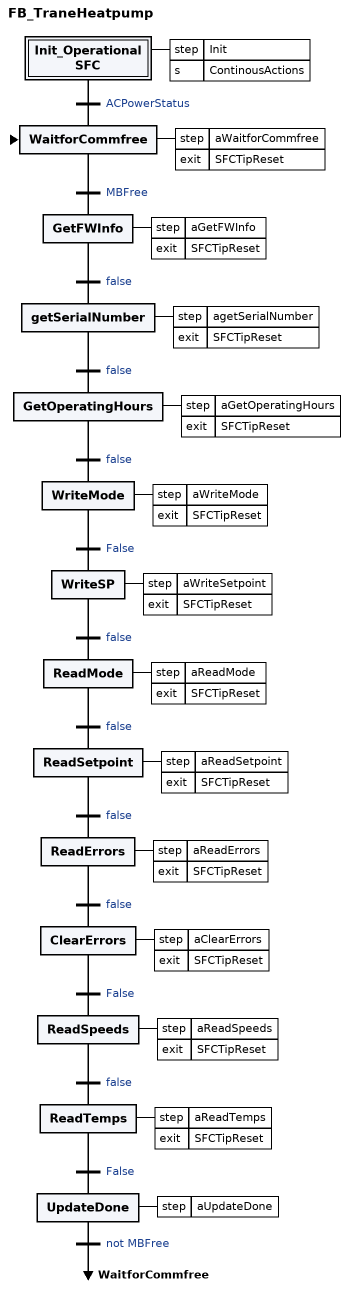
INITIAL_STEP Init_OperationalSFC:
    Init(N);  // step action
    ContinousActions(s);
END_STEP
TRANSITION FROM Init_OperationalSFC TO WaitforCommfree
    := ACPowerStatus;
END_TRANSITION
STEP WaitforCommfree:
    aWaitforCommfree(N);  // step action
    SFCTipReset(P0);  // exit action
END_STEP
TRANSITION FROM WaitforCommfree TO GetFWInfo
    := MBFree;
END_TRANSITION
STEP GetFWInfo:  // max time T#2S
    aGetFWInfo(N);  // step action
    SFCTipReset(P0);  // exit action
END_STEP
TRANSITION FROM GetFWInfo TO getSerialNumber
    := false;
END_TRANSITION
STEP getSerialNumber:  // max time T#2S
    agetSerialNumber(N);  // step action
    SFCTipReset(P0);  // exit action
END_STEP
TRANSITION FROM getSerialNumber TO GetOperatingHours
    := false;
END_TRANSITION
STEP GetOperatingHours:  // max time T#2S
    aGetOperatingHours(N);  // step action
    SFCTipReset(P0);  // exit action
END_STEP
TRANSITION FROM GetOperatingHours TO WriteMode
    := false;
END_TRANSITION
STEP WriteMode:  // max time T#2S
    aWriteMode(N);  // step action
    SFCTipReset(P0);  // exit action
END_STEP
TRANSITION FROM WriteMode TO WriteSP
    := False;
END_TRANSITION
STEP WriteSP:  // max time T#2S
    aWriteSetpoint(N);  // step action
    SFCTipReset(P0);  // exit action
END_STEP
TRANSITION FROM WriteSP TO ReadMode
    := false;
END_TRANSITION
STEP ReadMode:  // max time T#2S
    aReadMode(N);  // step action
    SFCTipReset(P0);  // exit action
END_STEP
TRANSITION FROM ReadMode TO ReadSetpoint
    := false;
END_TRANSITION
STEP ReadSetpoint:  // max time T#2S
    aReadSetpoint(N);  // step action
    SFCTipReset(P0);  // exit action
END_STEP
TRANSITION FROM ReadSetpoint TO ReadErrors
    := false;
END_TRANSITION
STEP ReadErrors:  // max time T#2S
    aReadErrors(N);  // step action
    SFCTipReset(P0);  // exit action
END_STEP
TRANSITION FROM ReadErrors TO ClearErrors
    := false;
END_TRANSITION
STEP ClearErrors:  // max time T#2S
    aClearErrors(N);  // step action
    SFCTipReset(P0);  // exit action
END_STEP
TRANSITION FROM ClearErrors TO ReadSpeeds
    := False;
END_TRANSITION
STEP ReadSpeeds:  // max time T#2S
    aReadSpeeds(N);  // step action
    SFCTipReset(P0);  // exit action
END_STEP
TRANSITION FROM ReadSpeeds TO ReadTemps
    := false;
END_TRANSITION
STEP ReadTemps:  // max time T#2S
    aReadTemps(N);  // step action
    SFCTipReset(P0);  // exit action
END_STEP
TRANSITION FROM ReadTemps TO UpdateDone
    := False;
END_TRANSITION
STEP UpdateDone:
    aUpdateDone(N);  // step action
END_STEP
TRANSITION FROM UpdateDone TO WaitforCommfree
    := not MBFree;
END_TRANSITION

ACTION aClearErrors:
IF b_resetErrors THEN
	
	Databuffer[0]	:= 0;
	
	MBMaster.WriteSingleRegister(
						UnitID 		:= 	HeatPumpID,
						MBAddr		:=	950,
						Quantity 	:= 	1,
						cbLength 	:= SIZEOF(Databuffer),
						pMemoryAddr	:=	ADR(Databuffer[0]),
						Execute		:=	ftrig_ModbusStartTrigger.Q,		
						);
						
	IF TransmissionDoneTrigger.q THEN
		IF NOT MBMaster.Error THEN
			b_resetErrors := FALSE;
		END_IF
		SFCTip := NOT SFCTip;
	END_IF

ELSE
	SFCTip := NOT SFCTip;
END_IF
END_ACTION

ACTION aGetFWInfo:
bMBActive := TRUE;

IF get.HeatPumpState = eHeatpumpState.Initializing THEN
	MBMaster.ReadRegs(	UnitID 		:= 	HeatPumpID,
						Quantity 	:= 	4,
						MBAddr		:=	1,
						cbLength 	:= 	SIZEOF(DataBuffer), //64
						pMemoryAddr	:=	ADR(DataBuffer),
						Execute		:=	ftrig_ModbusStartTrigger.Q,

						);
	

	IF TransmissionDoneTrigger.q THEN
		IF NOT MBMaster.Error AND MBmaster.cbRead = 8 THEN
			get.HeatpumpData.i_FW_Version 		:= 	WORD_TO_INT(DataBuffer[0]);
			get.HeatpumpData.i_FW_release 		:= 	WORD_TO_INT(DataBuffer[1]);
			get.HeatpumpData.w_FW_Subrelease 	:= 	DataBuffer[2];
			get.HeatpumpData.w_FW_creationDate	:=	DataBuffer[3];
			MBRetryCount := 0;	
			sfctip := TRUE;
		ELSE
			MBRetryCount := MBRetryCount + 1;

		END_IF
	END_IF
ELSE
	sfctip := NOT sfctip;
END_IF
END_ACTION

ACTION aGetOperatingHours:


MBMaster.ReadRegs(	UnitID 		:= 	HeatPumpID,
					Quantity 	:= 	1,
					MBAddr		:=	305,
					cbLength 	:= 	SIZEOF(Databuffer),
					pMemoryAddr	:=	ADR(DataBuffer),
					Execute		:=	ftrig_ModbusStartTrigger.Q,
					);



IF TransmissionDoneTrigger.q THEN
	IF NOT MBMaster.Error THEN
		//transmission done, process data
		
		//just use comp 1 for now. See if the others are even used
		//i think it will be a dual word value. But check later
		get.HeatpumpData.i_OperatingHours := WORD_TO_INT(DataBuffer[0]);
		
		//done, preset for next step
		MBRetryCount := 0;
	ELSE
		MBRetryCount := MBRetryCount + 1;
	END_IF
	sfctip := TRUE;
END_IF
END_ACTION

ACTION agetSerialNumber:

IF get.HeatPumpState = eHeatpumpState.Initializing THEN
	MBMaster.ReadRegs(	UnitID 		:= 	HeatPumpID,
						Quantity 	:= 	18,
						MBAddr		:=	80,
						cbLength 	:= 	SIZEOF(Databuffer),//32*2,
						pMemoryAddr	:=	ADR(DataBuffer),
						Execute		:=	ftrig_ModbusStartTrigger.Q,	
						);
	
	IF TransmissionDoneTrigger.q THEN
		IF NOT MBMaster.Error THEN
			FOR u_counter:=0 TO 17 BY 1 DO
				get.HeatpumpData.w_Serialnumber[u_counter]	:= 	DataBuffer[u_counter];
			END_FOR
			MBRetryCount := 0;
		
			sfctip := TRUE;
			get.HeatPumpState := eHeatpumpState.Standby;
		ELSE
			MBRetryCount := MBRetryCount + 1;
			
		END_IF
	END_IF
ELSE
	sfctip := NOT sfctip;
END_IF
END_ACTION

METHOD AllowMBComm : BOOL
VAR_INPUT
	b_AllowComm	:	Bool;
END_VAR
MBFree	:= b_AllowComm;
END_METHOD

ACTION aReadErrors:

MBMaster.ReadRegs(	UnitID 		:= 	HeatPumpID,
					Quantity 	:= 	7,
					MBAddr		:=	950,
					cbLength 	:= 	SIZEOF(Databuffer),
					pMemoryAddr	:=	ADR(DataBuffer),
					Execute		:=	ftrig_ModbusStartTrigger.Q,
					);

IF TransmissionDoneTrigger.q THEN
	IF NOT MBMaster.Error AND MBMaster.cbRead = 14 THEN
	
			ParseHeatPumpErrors(	w_Alarms1 := DataBuffer[0],
									w_Alarms2 := DataBuffer[1],
									w_Alarms3 := DataBuffer[2],
									w_Alarms4 := DataBuffer[3],
									w_Alarms5 := DataBuffer[4],
									w_Alarms6 := DataBuffer[5],
									w_Alarms7 := DataBuffer[6],
									Get := Get			
								);
			
			//done, preset for next step
			
			MBRetryCount := 0;

	ELSE
		MBRetryCount := MBRetryCount + 1;
				
	END_IF
	sfctip := TRUE;
END_IF
END_ACTION

ACTION aReadMode:

MBMaster.ReadRegs(	UnitID 		:= 	HeatPumpID,
					Quantity 	:= 	1,
					MBAddr		:=	200,
					cbLength 	:= 	SIZEOF(Databuffer),
					pMemoryAddr	:=	ADR(DataBuffer),
					Execute		:=	ftrig_ModbusStartTrigger.Q,
					);


IF TransmissionDoneTrigger.q THEN
	IF NOT MBMaster.Error THEN
	
		//transmission done, process data
		CASE DataBuffer[0] OF
			0:	get.HeatPumpState := eHeatpumpState.Standby;
			1:	get.HeatPumpState := eHeatpumpState.Active_Cooling;
			2:	get.HeatPumpState := eHeatpumpState.Active_Heating;
		END_CASE
		
		//done, preset for next step
		MBRetryCount := 0;

	ELSE
		MBRetryCount := MBRetryCount + 1;
		
	END_IF
	sfctip := TRUE;
END_IF
END_ACTION

ACTION aReadSetpoint:

//r_FanSpeedPCT			:	REAL;		//7000
//r_PumpSpeedPCT		:	REAL;		//7001

MBMaster.ReadRegs(	UnitID 		:= 	HeatPumpID,
					Quantity 	:= 	2,
					MBAddr		:=	7203,
					cbLength 	:= 	SIZEOF(Databuffer),
					pMemoryAddr	:=	ADR(DataBuffer),
					Execute		:=	ftrig_ModbusStartTrigger.Q,		
					);

IF TransmissionDoneTrigger.q THEN
	IF NOT MBMaster.Error THEN
	
		//transmission done, process data
		get.HeatpumpData.r_SetpointHeating	:=	DataBuffer[1]/10;
		get.HeatpumpData.r_SetpointCooling	:=	DataBuffer[0]/10;
		//done, preset for next step
		MBRetryCount := 0;
	ELSE
		MBRetryCount := MBRetryCount + 1;
	END_IF
	
	sfctip := TRUE;
END_IF
END_ACTION

ACTION aReadSpeeds:

//r_FanSpeedPCT			:	REAL;		//7000
//r_PumpSpeedPCT		:	REAL;		//7001

MBMaster.ReadRegs(	UnitID 		:= 	HeatPumpID,
					Quantity 	:= 	2,
					MBAddr		:=	7000,
					cbLength 	:= 	SIZEOF(Databuffer),
					pMemoryAddr	:=	ADR(DataBuffer),
					Execute		:=	ftrig_ModbusStartTrigger.Q,		
					);

IF TransmissionDoneTrigger.q THEN
	IF NOT MBMaster.Error THEN
		
		//transmission done, process data
		get.HeatpumpData.r_FanSpeedPCT		:=	WORD_TO_REAL(DataBuffer[0])/10;
		get.HeatpumpData.r_PumpSpeedPCT		:= 	WORD_TO_REAL(DataBuffer[1])/10;
		
		MBRetryCount := 0;
	ELSE
		MBRetryCount := MBRetryCount + 1;
	END_IF
	sfctip := TRUE;
END_IF
END_ACTION

ACTION aReadTemps:

(*
r_InletWaterTemp	:	REAL;		//400
r_OutletWaterTemp	:	REAL;		//401
r_HighPressure		:	REAL;		//406
r_LowPressure		:	REAL;		//414
r_CompInputTemp		:	REAL;		//422
r_OutdoorTemp		:	REAL;		//428
r_CompOutputTemp	:	REAL;		//433-435
ui_WaterFlowRate		:	uINT;		//444
*)

MBMaster.ReadRegs(	UnitID 		:= 	HeatPumpID,
					Quantity 	:= 	45,
					MBAddr		:=	400,
					cbLength 	:= 	SIZEOF(Databuffer),
					pMemoryAddr	:=	ADR(DataBuffer),
					Execute		:=	ftrig_ModbusStartTrigger.Q,		
					);


IF TransmissionDoneTrigger.q THEN
	IF NOT MBMaster.Error THEN
		
		//transmission done, process data
		get.HeatpumpData.r_InletWaterTemp		:=	INT_TO_REAL(DataBuffer[0])/10;
		get.HeatpumpData.r_OutletWaterTemp		:= 	INT_TO_REAL(DataBuffer[1])/10;
		get.HeatpumpData.r_HighPressure			:=	INT_TO_REAL(DataBuffer[6])/100;
		get.HeatpumpData.r_LowPressure			:= 	INT_TO_REAL(DataBuffer[14])/100;
		get.HeatpumpData.r_CompInputTemp		:=	INT_TO_REAL(DataBuffer[22])/10;
		get.HeatpumpData.r_OutdoorTemp			:= 	INT_TO_REAL(DataBuffer[28])/10;
		get.HeatpumpData.r_CompOutputTemp		:=	INT_TO_REAL(DataBuffer[33])/10;	//comp dischyarge 1 for now
		get.HeatpumpData.ui_WaterFlowRate			:= 	DataBuffer[44];
		
		MBRetryCount := 0;
	ELSE
		MBRetryCount := MBRetryCount + 1;
	END_IF
	sfctip := TRUE;
END_IF
END_ACTION

ACTION aUpdateDone:
SFCTip := FALSE;
bMBActive := FALSE;
END_ACTION

ACTION aWaitforCommfree:
//SFCTip := FALSE;
//b_EnableTransmission	:= FALSE;
//ModbusStartTrigger(clk := b_EnableTransmission);
END_ACTION

ACTION aWriteMode:
//SFCTip := FALSE;


//b_EnableTransmission	:= TRUE;
//ModbusStartTrigger(clk := b_EnableTransmission);

Databuffer[0]	:= RequestedSetpoint.OperatingMode;	//set operating mode for write
Databuffer[1]	:= 3;								//enable write registers

MBMaster.WriteRegs ( 
					UnitID 		:= 	HeatPumpID,
					Quantity 	:= 	2,
					MBAddr		:=	7200,
					cbLength 	:= 	SIZEOF(Databuffer),
					pMemoryAddr	:=	ADR(Databuffer),
					Execute		:=	ftrig_ModbusStartTrigger.Q,		
					);
				
IF TransmissionDoneTrigger.q THEN
	IF NOT MBMaster.Error THEN
				
		MBRetryCount := 0;
	ELSE
		MBRetryCount := MBRetryCount + 1;
	END_IF
	sfctip := TRUE;
END_IF
END_ACTION

ACTION aWriteSetpoint:

CASE RequestedSetpoint.OperatingMode OF				//Update setpoint depending on mode
	eHeatPumpMode.Cooling:
		Databuffer[0]	:= REAL_TO_WORD(LIMIT(50, ((RequestedSetpoint.Setpoint)*10), 230));
		Databuffer[1]	:= REAL_TO_WORD(Get.HeatpumpData.r_SetpointHeating*10);
	eHeatPumpMode.Heating:
		Databuffer[0]	:= REAL_TO_WORD(Get.HeatpumpData.r_SetpointCooling*10);
		Databuffer[1]	:= REAL_TO_WORD(LIMIT(250, ((RequestedSetpoint.Setpoint)*10), 550));
	eHeatPumpMode.Standby:
		Databuffer[0]	:= REAL_TO_WORD(Get.HeatpumpData.r_SetpointCooling*10);
		Databuffer[1]	:= REAL_TO_WORD(Get.HeatpumpData.r_SetpointHeating*10);	
END_CASE

MBMaster.WriteRegs (
		UnitID 		:= 	HeatPumpID,
		Quantity 	:= 	2,
		MBAddr		:=	7203,
		cbLength 	:= 	SIZEOF(Databuffer),
		pMemoryAddr	:=	ADR(Databuffer),
		Execute		:=	ftrig_ModbusStartTrigger.Q,		
);



IF TransmissionDoneTrigger.q THEN
	IF NOT MBMaster.Error THEN
		//done, preset for next step

		MBRetryCount := 0;;
	ELSE
		MBRetryCount := MBRetryCount + 1;
	END_IF
	sfctip := TRUE;
END_IF
END_ACTION

ACTION ContinousActions:
//sfctip := False;
ton_modbusStuckTrigger(in := NOT ton_modbusStuckTrigger.q AND NOT TP_ModbusStartTriggerDelay.q);
TP_ModbusStartTriggerDelay(IN := NOT MBMaster.BUSY AND NOT ton_modbusStuckTrigger.q );
ftrig_ModbusStartTrigger(clk := TP_ModbusStartTriggerDelay.Q);

IF SFCError THEN
	SFCError := FALSE;
	get.Events.b_CommWarning := TRUE;
END_IF

IF NOT ACPowerStatus THEN
	IF get.HeatPumpState <> eHeatpumpstate.OFF THEN
		get.HeatPumpState := eHeatpumpState.OFF;
		SFCReset := TRUE;
	END_IF
END_IF


//safeguard, should the sfc get stuck, heatpumpsystem can revoke MB rights and SFC resets.
//IF NOT MBfree AND bMBActive AND NOT MBMaster.BUSY THEN
//	SFCReset := TRUE;
//END_IF 

IF ACPowerStatus AND get.HeatPumpState = eHeatpumpState.OFF THEN
	get.HeatPumpState := eHeatpumpState.Initializing;
END_IF

HeatpumpPreheatControl();


//reset mb master if stuck in busy
ton_MBBUSYTimeOut(IN := MBmaster.BUSY);
IF ton_MBBUSYTimeOut.Q THEN
	MBMaster.ReadRegs();
	MBMaster.WriteRegs();
	MBMaster.WriteSingleRegister();
END_IF

//Reset heatpump when error occurs, but after a bit of cooldown time.
//Maybe add a functionality to stop trying after x tries to prevent continuous reset cycles
Ton_ErrorTimer(in := get.Events.b_CompressorError OR 
					get.Events.b_FanError OR 
					get.Events.b_PressureError OR 
					get.Events.b_WaterTempError OR 
					get.Events.b_PumpError );
IF Ton_ErrorTimer.Q THEN
	b_resetErrors := TRUE;
END_IF

TransmissionDoneTrigger(clk := MBMaster.Busy);
MBMaster.Timeout		:= st_params.t_ModbusTimeOut;		

get.Events.b_CommWarning := MBRetryCount > st_params.i_modbusRetries;
END_ACTION

METHOD EMStop : BOOL
RequestedSetpoint.OperatingMode := eHeatpumpMode.Standby;
b_Emstop := TRUE;
EMstop := TRUE;
END_METHOD

METHOD GetDiagnostics 
VAR_IN_OUT
	AddError		: ARRAY [*] OF FB_AddErrorST;
	a_ActiveEvents	: ARRAY [*] OF ST_ErrorStruct;
	w_Index			: WORD;
END_VAR

VAR_OUTPUT
	b_errorActive	: BOOL;
	b_warningActive	: BOOL;
END_VAR

VAR
	by_errCt	: BYTE;
	by_warnCt	: BYTE;
END_VAR
	(*Modbus comm fault*)	AddError[w_Index](
			b_ErrorTrig			:= Get.Events.b_commwarning,
			out_ST_Error			:= a_ActiveEvents[w_Index],
			w_ErrorID				:= 30 + ((HeatPumpID-1)*10),
			e_ObjectID				:= e_ID,
			s_Message				:= 'Modbus communication fault',
			e_sev					:= eSeverity.Warning,	
			b_AutoClear			:= TRUE,
			t_TriggerTime		:=	T#60s,
			//in_e_ErrAckAccess		:= TRUE,
			);
		w_Index := w_Index +1;
		
	(*Heatpump Compressor fault*)	AddError[w_Index](
			b_ErrorTrig			:= Get.Events.b_CompressorError,
			out_ST_Error			:= a_ActiveEvents[w_Index],
			w_ErrorID				:= 31 + ((HeatPumpID-1)*10),
			s_Message				:= concat('Compressor fault', sCompressorErrorText),
			e_sev					:= eSeverity.Warning,	
			b_AutoClear			:= FALSE,
			t_TriggerTime		:=	T#1S,
			//in_e_ErrAckAccess		:= TRUE,
			);
		w_Index := w_Index +1;
	
	
	(*Heatpump Fan fault*)			AddError[w_Index](
			b_ErrorTrig			:= Get.Events.b_FanError,
			out_ST_Error			:= a_ActiveEvents[w_Index],
			w_ErrorID				:= 32 + ((HeatPumpID-1)*10),
			s_Message				:= 'Fan fault',
			e_sev					:= eSeverity.Warning,	
			b_AutoClear			:= FALSE,
			t_TriggerTime		:=	T#1S,
			//in_e_ErrAckAccess		:= TRUE,
			);
		w_Index := w_Index +1;
		
	(*HHeatpump Internal IO fault*)		AddError[w_Index](
			b_ErrorTrig			:= Get.Events.b_IOError ,
			out_ST_Error			:= a_ActiveEvents[w_Index],
			w_ErrorID				:= 33 + ((HeatPumpID-1)*10),
			s_Message				:= 'internal IO fault',
			e_sev					:= eSeverity.Warning,	
			b_AutoClear			:= FALSE,
			t_TriggerTime		:=	T#1S,
			//in_e_ErrAckAccess		:= TRUE,
			);
		w_Index := w_Index +1;
		
	(*Heatpump pressure fault*)		AddError[w_Index](
			b_ErrorTrig			:= Get.Events.b_PressureError,
			out_ST_Error			:= a_ActiveEvents[w_Index],
			w_ErrorID				:= 34 + ((HeatPumpID-1)*10),
			s_Message				:= concat('pressure fault', sPressureErrorText),
			e_sev					:= eSeverity.Warning,	
			b_AutoClear			:= FALSE,
			t_TriggerTime		:=	T#1S,
			//in_e_ErrAckAccess		:= TRUE,
			);
		w_Index := w_Index +1;

	(*Heatpump Probe fault*)		AddError[w_Index](
			b_ErrorTrig			:= Get.Events.b_ProbeError,
			out_ST_Error			:= a_ActiveEvents[w_Index],
			w_ErrorID				:= 35 + ((HeatPumpID-1)*10),
			s_Message				:= 'probe fault',
			e_sev					:= eSeverity.Warning,	
			b_AutoClear			:= FALSE,
			t_TriggerTime		:=	T#1S,
			//in_e_ErrAckAccess		:= TRUE,
			);
		w_Index := w_Index +1;	

	(*Heatpump Pump fault*)			AddError[w_Index](
			b_ErrorTrig			:= Get.Events.b_PumpError,
			out_ST_Error			:= a_ActiveEvents[w_Index],
			w_ErrorID				:= 36 + ((HeatPumpID-1)*10),
			s_Message				:= concat('pump fault', sPumpErrorText),
			e_sev					:= eSeverity.Warning,	
			b_AutoClear			:= FALSE,
			t_TriggerTime		:=	T#1S,
			//in_e_ErrAckAccess		:= TRUE,
			);
		w_Index := w_Index +1;	

	(*Heatpump valve fault*)			AddError[w_Index](
			b_ErrorTrig			:= Get.Events.b_ValveError,
			out_ST_Error			:= a_ActiveEvents[w_Index],
			w_ErrorID				:=37 + ((HeatPumpID-1)*10),
			s_Message				:= 'valve fault',
			e_sev					:= eSeverity.Warning,	
			b_AutoClear			:= FALSE,
			t_TriggerTime		:=	T#1S,
			//in_e_ErrAckAccess		:= TRUE,
			);
		w_Index := w_Index +1;	

	(*Heatpump Water temperature error*)			AddError[w_Index](
			b_ErrorTrig			:= Get.Events.b_WaterTempError,
			out_ST_Error			:= a_ActiveEvents[w_Index],
			w_ErrorID				:= 38 + ((HeatPumpID-1)*10),
			s_Message				:= concat('water temperature error', sWaterTempErrorText),
			e_sev					:= eSeverity.Warning,	
			b_AutoClear			:= FALSE,
			t_TriggerTime		:=	T#1S,
			//in_e_ErrAckAccess		:= TRUE,
			);
		w_Index := w_Index +1;		
		
	(*Heatpump Preheating active*)			AddError[w_Index](
			b_ErrorTrig				:= Get.Events.b_HeatpumpPreheatingActive,
			out_ST_Error			:= a_ActiveEvents[w_Index],
			w_ErrorID				:= 39 + ((HeatPumpID-1)*10),
			s_Message				:= concat('Heatpump preheating active for ', TO_STRING(t_RemainingPreheatingTime)),
			e_sev					:= eSeverity.Info,	
			b_AutoClear				:= TRUE,
			);
		w_Index := w_Index +1;
END_METHOD

METHOD PRIVATE HeatpumpPreheatControl : BOOL
VAR
	b_PreheatingRequired	:	BOOL;
END_VAR

VAR_INST
	ton_PreheatingTimer	:	Ton;
END_VAR
//enable operation
ton_PreheatingTimer(IN:= ACPowerStatus, PT:= TO_TIME(st_params.dw_HeatpumpOperationDelay*1000*60));
b_PreheatingRequired := ((DT_TO_INT(GVL.dt_SystemDateTime) - DT_TO_INT(dt_LastHPOperationTime))/60) > st_params.i_SkipHPPreheatingTime;

t_RemainingPreheatingTime := ton_PreheatingTimer.PT - ton_preheatingTimer.ET;

IF ton_PreheatingTimer.Q THEN
	dt_LastHPOperationTime := GVL.dt_SystemDateTime;
	t_RemainingPreheatingTime := T#0ms;
END_IF

get.Events.b_HeatpumpPreheatingActive := b_PreheatingRequired AND ACPowerStatus ;
END_METHOD

ACTION Init:
get.HeatPumpState := eHeatpumpstate.OFF;
bmbActive := FALSE;
SFCReset := false;
END_ACTION

METHOD MBCommBusy : BOOL
VAR_INPUT
END_VAR
MBCommBusy := bMBActive;
END_METHOD

METHOD ParseHeatPumpErrors : BOOL
VAR_INPUT
	w_Alarms1	:	WORD;
	w_Alarms2	:	WORD;
	w_Alarms3	:	WORD;
	w_Alarms4	:	WORD;
	w_Alarms5	:	WORD;
	w_Alarms6	:	WORD;
	w_Alarms7	:	WORD;
END_VAR		


VAR_IN_OUT
	get	:	ST_HeatPump_Get;	
END_VAR
get.events.b_ProbeError		:=	WORD_TO_BOOL(w_Alarms3) OR WORD_TO_BOOL(w_Alarms4) OR w_Alarms5.0;

get.events.b_PressureError		:=	w_Alarms1.0 OR	//E001: High Pressure
									w_Alarms1.1 OR //E002: Low Pressure
									w_Alarms2.3;	//E020: Inverted Pressure Transducers
									
sPressureErrorText := '';
IF get.events.b_PressureError THEN
	sPressureErrorText := concat(sPressureErrorText, SEL(w_Alarms1.0, '', ' E001'));
	sPressureErrorText := concat(sPressureErrorText, SEL(w_Alarms1.1, '', ' E002'));
	sPressureErrorText := concat(sPressureErrorText, SEL(w_Alarms2.3, '', ' E020'));
END_IF
									
get.events.b_CompressorError	:=	w_Alarms1.2 OR //E003: Compressor overheated
									w_Alarms1.7 OR //E008: Compressor underspeed
									w_Alarms1.8 OR	//E009: High disch temp
									w_Alarms1.12 OR //E013: Comp2 Overheated
									w_Alarms2.2 OR	//E019: CP2 High disch temp
									w_Alarms2.6 OR	//E023: Comp3 Overheated
									w_Alarms5.1 OR //'E801: Link Inverter1',
									w_Alarms5.2 OR //'E802: Link Inverter2',
									w_Alarms5.3 OR //'E803: Link Inverter3',
									w_Alarms5.4 OR //'E851: HWfault Inverter1',
									w_Alarms5.5 OR //'E852: HWfault Inverter2',
									w_Alarms5.6 OR //'E853: HWfault Inverter3',
									w_Alarms5.7 OR //'E861: OverCurrent Inv1',
									w_Alarms5.8 OR //'E862: OverCurrent Inv2',
									w_Alarms5.9 OR //'E863: OverCurrent Inv3',
									w_Alarms5.10 OR //'E871: High Temp Inv1',
									w_Alarms5.11 OR //'E872: High Temp Inv2',
									w_Alarms5.12 OR //'E873: High Temp Inv3',
									w_Alarms5.13 OR //'E881: Bad Voltage Inv1',
									w_Alarms5.14 OR //'E882: Bad Voltage Inv2',
									w_Alarms5.15 OR //'E883: Bad Voltage Inv3',
									w_Alarms6.0 OR //E891: Phase Seq Inv1',
									w_Alarms6.1 OR //'E892: Phase Seq Inv2',
									w_Alarms6.2 OR //'E893: Phase Seq Inv3',
									w_Alarms6.3 OR //'E901: Model err Inv1',
									w_Alarms6.4 OR //'E902: Model err Inv2',
									w_Alarms6.5 OR //'E903: Model err Inv3',
									w_Alarms6.6 OR //'E911: Ovl error Inv1',
									w_Alarms6.7 OR //'E9112: Ovl error Inv2',
									w_Alarms6.8 OR //'E913: Ovl error Inv3',
									w_Alarms6.9 OR //'E921: Overc PFC Inv1',
									w_Alarms6.10 OR //'E922: Overc PFC Inv2',
									w_Alarms6.11 OR //'E923: Overc PFC Inv3',
									w_Alarms6.12 OR //'E931: Int Com ERR Inv1',
									w_Alarms6.13 OR //'E932: Int Com ERR Inv2',
									w_Alarms6.14 OR //'E933: Int Com ERR Inv3',
									w_Alarms6.15 OR //'E941: Fault PFC Inv1',
									w_Alarms7.0 OR //E942: Fault PFC Inv2
									w_Alarms7.1 OR //'E943: Fault PFC Inv3',
									w_Alarms7.2 OR //'E951: Probe error Inv1',
									w_Alarms7.3 OR //'E952: Probe error Inv2',
									w_Alarms7.4 OR //'E953: Probe error Inv3',
									w_Alarms7.5 OR //'E961: Abnormal Cond Inv1',
									w_Alarms7.6 OR //'E962: Abnormal Cond Inv2',
									w_Alarms7.7 OR //'E963: Abnormal Cond Inv3',
									w_Alarms7.8 OR //'E971: Inv1 Eeprom Error',
									w_Alarms7.9 OR //'E972: Inv2 Eeprom Error',
									w_Alarms7.10 OR //'E973: Inv3 Eeprom Error',
									w_Alarms7.11;	//E029: CP3 High disch temp

sCompressorErrorText := '';
IF get.events.b_CompressorError THEN
	sCompressorErrorText := concat(sCompressorErrorText, SEL(w_Alarms1.2, '', ' E003'));
	sCompressorErrorText := concat(sCompressorErrorText, SEL(w_Alarms1.7, '', ' E008'));
	sCompressorErrorText := concat(sCompressorErrorText, SEL(w_Alarms1.8, '', ' E009'));
	sCompressorErrorText := concat(sCompressorErrorText, SEL(w_Alarms1.12, '', ' E013'));
	sCompressorErrorText := concat(sCompressorErrorText, SEL(w_Alarms2.2, '', ' E019'));
	sCompressorErrorText := concat(sCompressorErrorText, SEL(w_Alarms2.6, '', ' E023'));
	sCompressorErrorText := concat(sCompressorErrorText, SEL(w_Alarms5.1, '', ' E801'));
	sCompressorErrorText := concat(sCompressorErrorText, SEL(w_Alarms5.2, '', ' E802'));
	sCompressorErrorText := concat(sCompressorErrorText, SEL(w_Alarms5.3, '', ' E803'));
	sCompressorErrorText := concat(sCompressorErrorText, SEL(w_Alarms5.4, '', ' E851'));
	sCompressorErrorText := concat(sCompressorErrorText, SEL(w_Alarms5.5, '', ' E852'));
	sCompressorErrorText := concat(sCompressorErrorText, SEL(w_Alarms5.6, '', ' E853'));
	sCompressorErrorText := concat(sCompressorErrorText, SEL(w_Alarms5.7, '', ' E861'));
	sCompressorErrorText := concat(sCompressorErrorText, SEL(w_Alarms5.8, '', ' E862'));
	sCompressorErrorText := concat(sCompressorErrorText, SEL(w_Alarms5.9, '', ' E863'));
	sCompressorErrorText := concat(sCompressorErrorText, SEL(w_Alarms5.10, '', ' E871'));
	sCompressorErrorText := concat(sCompressorErrorText, SEL(w_Alarms5.11, '', ' E872'));
	sCompressorErrorText := concat(sCompressorErrorText, SEL(w_Alarms5.12, '', ' E873'));
	sCompressorErrorText := concat(sCompressorErrorText, SEL(w_Alarms5.13, '', ' E881'));
	sCompressorErrorText := concat(sCompressorErrorText, SEL(w_Alarms5.14, '', ' E882'));
	sCompressorErrorText := concat(sCompressorErrorText, SEL(w_Alarms5.15, '', ' E883'));
	sCompressorErrorText := concat(sCompressorErrorText, SEL(w_Alarms6.0 , '', ' E891'));
	sCompressorErrorText := concat(sCompressorErrorText, SEL(w_Alarms6.1 , '', ' E892'));
	sCompressorErrorText := concat(sCompressorErrorText, SEL(w_Alarms6.2 , '', ' E893'));
	sCompressorErrorText := concat(sCompressorErrorText, SEL(w_Alarms6.3 , '', ' E901'));
	sCompressorErrorText := concat(sCompressorErrorText, SEL(w_Alarms6.4 , '', ' E902'));
	sCompressorErrorText := concat(sCompressorErrorText, SEL(w_Alarms6.5 , '', ' E903'));
	sCompressorErrorText := concat(sCompressorErrorText, SEL(w_Alarms6.6 , '', ' E911'));
	sCompressorErrorText := concat(sCompressorErrorText, SEL(w_Alarms6.7 , '', ' E912'));
	sCompressorErrorText := concat(sCompressorErrorText, SEL(w_Alarms6.8 , '', ' E913'));
	sCompressorErrorText := concat(sCompressorErrorText, SEL(w_Alarms6.9 , '', ' E921'));
	sCompressorErrorText := concat(sCompressorErrorText, SEL(w_Alarms6.10, '', ' E922'));
	sCompressorErrorText := concat(sCompressorErrorText, SEL(w_Alarms6.11, '', ' E923'));
	sCompressorErrorText := concat(sCompressorErrorText, SEL(w_Alarms6.12, '', ' E931'));
	sCompressorErrorText := concat(sCompressorErrorText, SEL(w_Alarms6.13, '', ' E932'));
	sCompressorErrorText := concat(sCompressorErrorText, SEL(w_Alarms6.14, '', ' E933'));
	sCompressorErrorText := concat(sCompressorErrorText, SEL(w_Alarms6.15, '', ' E941'));
	sCompressorErrorText := concat(sCompressorErrorText, SEL(w_Alarms7.0 , '', ' E942'));
	sCompressorErrorText := concat(sCompressorErrorText, SEL(w_Alarms7.1 , '', ' E943'));
	sCompressorErrorText := concat(sCompressorErrorText, SEL(w_Alarms7.2 , '', ' E951'));
	sCompressorErrorText := concat(sCompressorErrorText, SEL(w_Alarms7.3 , '', ' E952'));
	sCompressorErrorText := concat(sCompressorErrorText, SEL(w_Alarms7.4 , '', ' E953'));
	sCompressorErrorText := concat(sCompressorErrorText, SEL(w_Alarms7.5 , '', ' E961'));
	sCompressorErrorText := concat(sCompressorErrorText, SEL(w_Alarms7.6 , '', ' E962'));
	sCompressorErrorText := concat(sCompressorErrorText, SEL(w_Alarms7.7 , '', ' E963'));
	sCompressorErrorText := concat(sCompressorErrorText, SEL(w_Alarms7.8 , '', ' E971'));
	sCompressorErrorText := concat(sCompressorErrorText, SEL(w_Alarms7.9 , '', ' E972'));
	sCompressorErrorText := concat(sCompressorErrorText, SEL(w_Alarms7.10, '', ' E973'));
	sCompressorErrorText := concat(sCompressorErrorText, SEL(w_Alarms7.11, '', ' E029'));
END_IF
								
get.events.b_ValveError		:=		w_Alarms2.11; //E041: Incongruent temps;


get.events.b_FanError			:=	w_Alarms1.2 OR //E004: Fan Overheated	
									w_Alarms1.13 OR //E014: Fan2 Overheated 
									w_Alarms2.7;	//E024: Fan3 Overheated					

get.events.b_PumpError			:=	w_Alarms1.5 OR	 	//E006: Lack of flow
									w_Alarms1.15 OR 	//E016: Pump Overheated
									w_Alarms2.9;		//E026: Pump2 Overheated

sPumpErrorText := '';
IF get.events.b_PumpError THEN
	sPumpErrorText := concat(sPumpErrorText, SEL(w_Alarms1.5, '', ' E006'));
	sPumpErrorText := concat(sPumpErrorText, SEL(w_Alarms1.15, '', ' E016'));
	sPumpErrorText := concat(sPumpErrorText, SEL(w_Alarms2.9, '', ' E026'));		
END_IF						
									
get.events.b_WaterTempError		:=	w_Alarms2.1 OR	//E018: OverTemperature
									w_Alarms1.4;	//E005: Frost

sWaterTempErrorText := '';									
IF get.events.b_WaterTempError THEN
	sWaterTempErrorText := concat(sWaterTempErrorText, SEL(w_Alarms1.5, '', ' E018'));
	sWaterTempErrorText := concat(sWaterTempErrorText, SEL(w_Alarms1.15, '', ' E005'));	
END_IF		


									
get.events.b_IOError			:=	w_Alarms2.14 OR 	//E101: IOMod1 Disconnected
									w_Alarms2.15; 		//E102: IOMod2 Disconnected
END_METHOD

METHOD Reset : BOOL
//until restarting the heatpump we don't know if errors are gone. So clear them for now.

get.Events.b_CompressorError := FALSE;
get.Events.b_FanError := FALSE;
get.Events.b_IOError := FALSE;
get.Events.b_PressureError := FALSE;
get.Events.b_ProbeError := FALSE;
get.Events.b_PumpError := FALSE;
get.Events.b_ValveError := FALSE;
get.Events.b_WaterTempError := FALSE;
b_Emstop := FALSE;

Reset := TRUE;
END_METHOD

METHOD Setpoint : BOOL
VAR_INPUT
	OperatingMode	:	eHeatpumpMode	:= 	eHeatpumpMode.Standby;
	Temperature		: 	REAL			:=	18;
END_VAR
IF get.HeatPumpState >= eHeatpumpstate.Standby AND 
	NOT get.Events.b_HeatpumpPreheatingActive AND 
	NOT b_EMstop THEN
	RequestedSetpoint.Setpoint		:= Temperature;
	RequestedSetpoint.OperatingMode := OperatingMode;
ELSE
	RequestedSetpoint.OperatingMode := eHeatPumpMode.Standby;
	RequestedSetpoint.Setpoint		:= 18.0;
END_IF

get.Setpoint := RequestedSetpoint.Setpoint;
END_METHOD

ACTION SFCTipReset:
SFCTip := FALSE;
END_ACTION

END_FUNCTION_BLOCK

// ---- POUs/Functions-FBs-Programs/_generalFunctions/fb_MovingAverage.TcPOU
FUNCTION_BLOCK fb_MovingAverage
VAR_INPUT
	IN 		: REAL;
	length	: UINT;
	enable 	: BOOL;
END_VAR
VAR_OUTPUT
	Q : REAL;
END_VAR
VAR
	r_Sumvalue		: REAL;
	ui_Index		: UINT; 
END_VAR

IF enable THEN
	r_Sumvalue := r_sumvalue + IN;
	ui_Index := ui_index +1;
	
	IF ui_index > length THEN
		r_Sumvalue := r_Sumvalue - Q * (ui_index - length +1);
		ui_index := length - 1; 
	END_IF
	
	Q := r_Sumvalue / MAX(1, ui_Index); 
ELSE
	Q := IN;
	r_Sumvalue := 0;
	ui_Index := 0;
END_IF

END_FUNCTION_BLOCK

// ---- POUs/Objects/CoolingSystem/FB_CoolingSystem_IO.TcPOU
FUNCTION_BLOCK FB_CoolingSystem_IO
VAR_IN_OUT CONSTANT
	st_params					: ST_Coolingsystem_params;
END_VAR

VAR_INPUT
	b_24VDCavailable			: BOOL;
	b_400Vavailable				: BOOL;
	b_inverterRunning			: BOOL;
END_VAR

VAR_OUTPUT
	r_CoolantPressure			: REAL;
	r_CoolantIdlePressure		: REAL;
	r_CoolantTemperature		: REAL;
END_VAR

VAR
	Inputs							AT %I*	:	ST_CoolingSystem_Inputs;
	Outputs							AT %Q* 	:	ST_CoolingSystem_Outputs;
	
	BattValveDelayTimer			: TON;
	FancoilValveDelayTimer		: TON;
	InvValveDelayTimer			: TON;
	
	DCPumpState					:	ePumpState;
	ACPumpState					:	ePumpState;
END_VAR

VAR_IN_OUT
	Events				: 	ST_CoolingSystem_Events; 
END_VAR

GetCoolantData(
	Pwarning := st_params.r_MinimumSystemBasePressureWarningLevel,
	PError := st_params.r_MinimumSystemBasePressureErrorLevel,
	PHyst := st_params.r_PressureHysteresis);

//Set events
FancoilValveDelayTimer(
	IN := (Outputs.BattLoopValveClose AND b_24VDCavailable) = Inputs.BattLoopValveFB,
	PT := INT_TO_TIME(st_params.i_MaximumValveOperatingTime*1000),
	Q => Events.b_BattLoopValveStuck);

InvValveDelayTimer(
	IN := (Outputs.InvLoopValveClose AND b_24VDCavailable) = Inputs.InvLoopValveFB,
	PT := INT_TO_TIME(st_params.i_MaximumValveOperatingTime*1000),
	Q => Events.b_InverterLoopValveStuck);
	
BattValveDelayTimer(
	IN := (Outputs.FancoilLoopValveClose AND b_24VDCavailable) = Inputs.FancoilLoopValveFB,
	PT := INT_TO_TIME(st_params.i_MaximumValveOperatingTime*1000),
	Q => Events.b_FancoilLoopValveStuck);

//400V fuse feedback
Events.b_CoolingSystemFuseFailure := NOT Inputs.CoolingSystem400VFuseFB;

//
CoolantPressureOK();
IF DCPumpState = ePumpState.Stopping THEN
	DCPumpOff(FALSE);
END_IF

METHOD PRIVATE ACPumpOff : BOOL
VAR_INPUT
END_VAR
outputs.ACPumpEnable := FALSE;
ACPumpState := ePumpState.Off;
Events.b_ACwaterPumpTimeOut :=  FALSE;

ACPumpOff := NOT outputs.ACPumpEnable;
END_METHOD

METHOD PRIVATE ACPumpOn : BOOL
VAR_INPUT
END_VAR

VAR_INST
	StartupPressureBaseValue	:	REAL;

	ton_StartupRetryTimer		: 	TON := (PT := T#15S);
	Ton_StartupFailedTimer		:	TON := (PT := T#1M);
	TP_PumpRetryDelay			:	Tp := (Pt := T#3S);
	rTrig_PumpStarted			:	r_Trig;
	
	//ACPump feedback comes up before pump is fully running
	TON_ACPumpFeedbackDelay		:	TON := (Pt := T#5S);
	
	b_test		:	BOOL;
END_VAR
Tp_PumpRetryDelay(IN := ton_StartupRetryTimer.Q);
ton_StartupRetryTimer(IN:= Outputs.ACPumpEnable);
Ton_StartupFailedTimer(IN:= ACPumpState = ePumpState.Starting);

TON_ACPumpFeedbackDelay(in:=inputs.ACPumpFB);

//Take reference value before pump starts
rTrig_PumpStarted(clk := outputs.ACPumpEnable);
IF rTrig_PumpStarted.Q THEN
	StartupPressureBaseValue := r_CoolantPressure;
END_IF

CASE ACPumpState OF
	ePumpState.Off:
		outputs.ACPumpEnable := FALSE;
		IF b_400VAvailable THEN
			ACPumpState := ePumpState.Starting;
		END_IF
		
	ePumpState.Starting:
		//enable pump power unless waiting for a retry
		outputs.ACPumpEnable := NOT TP_PumpRetryDelay.Q;
			
		//Switch to running mode if presure rise is reached
		IF ((r_CoolantPressure - StartupPressureBaseValue) > st_params.r_MainPumpMinimumPressure) OR TON_ACPumpFeedbackDelay.q THEN
			ACPumpState := ePumpState.Running;
		END_IF


		IF Ton_StartupFailedTimer.Q THEN
			Events.b_ACwaterPumpTimeOut := TRUE;
			ACPumpState := ePumpState.Off;
		END_IF
	
	ePumpState.Running:
		outputs.ACPumpEnable := TRUE;
		IF NOT b_400VAvailable THEN
			ACPumpState := ePumpState.OFF;
		END_IF
		
		IF st_params.b_MainPumpFbInstalled AND NOT inputs.ACPumpFb THEN
			ACPumpState := ePumpState.OFF;
		END_IF
		
		//METHOD NOT tested yet, so uncommented FOR now
		//IF NOT CoolantPressureOK() THEN
		//	ACPumpState := ePumpState.OFF;
		//END_IF

END_CASE


ACPumpOn	:=	ACPumpState = ePumpState.Running;
END_METHOD

METHOD BatteryCooling : BOOL
VAR_INPUT
END_VAR

VAR_INST
	InvLoopFb		: BOOL;
END_VAR

BatteryCooling := DisableInverterLoop() AND ACPumpON();
END_METHOD

METHOD CoolantPressureOK : BOOL
VAR_INPUT
END_VAR

VAR_INST
	PumpPressureDataArray	:	ARRAY[1..600] OF float;
	PumpPressure			:	fb_CTRL_MOVING_AVERAGE;
	PumpPressureParams		:	ST_CTRL_MOVING_AVERAGE_PARAMS := (	tCtrlCycleTime := T#500MS, 
																	tTaskCycleTime := T#10MS, 
																	nSamplesToFilter:=600);
																
	ftrig_BattValveOpening		:	f_trig;
	ftrig_FancoilValveOpening	:	f_trig;
	tp_ignorePressureDrop		:	TP := (PT := T#5S); 
END_VAR
ftrig_BattValveOpening(clk := Outputs.BattLoopValveClose);
ftrig_FancoilValveOpening(clk := Outputs.FancoilLoopValveClose);
tp_ignorePressureDrop(in:= ftrig_FancoilValveOpening.Q OR ftrig_BattValveOpening.q);

PumpPressureParams.pWorkArray_ADR := ADR(PumpPressureDataArray);
PumpPressureParams.nWorkArray_SIZEOF := SIZEOF(PumpPressureDataArray);

PumpPressure(	fIn := r_CoolantPressure, 
				eMode := E_CTRL_Mode.eCTRL_MODE_ACTIVE, 
				stParams := PumpPressureParams,
				fManSyncValue := r_CoolantPressure, 
				bSync := tp_ignorePressureDrop.Q);
				
CoolantPressureOK := ABS(PumpPressure.fOut - r_CoolantPressure) < st_params.AllowedCoolantPressureDrop;
END_METHOD

METHOD PRIVATE DCPumpOff : BOOL
VAR_INPUT
	force : BOOL;
END_VAR

VAR_INST
	t_Offdelay : TIME :=  T#5M;
	tof_PumpShutdownDelay	: TOF;
END_VAR
tof_PumpShutdownDelay(in:= DCPumpState = ePumpState.Running, PT := SEL(force, t_Offdelay, T#0S));

CASE DCPumpState OF
	ePumpState.Running, ePumpState.Starting:
		IF ACPumpState = ePumpState.Running THEN
			DCPumpState := ePumpState.Stopping;
		ELSE
			DCPumpState := ePumpState.off;
		END_IF
		
	ePumpState.Stopping:
		IF NOT tof_PumpShutdownDelay.q THEN
			DCPumpState := ePumpState.Off;
		END_IF

	ePumpState.off:
	outputs.DCPumpEnable := FALSE;
END_CASE

Events.b_DCpumpTimeout := FALSE;
Events.b_DCpumpPressureFault := FALSE;
DCpumpOff := DCPumpState = ePumpState.Off;
END_METHOD

METHOD PRIVATE DCPumpOn : BOOL

VAR_INST
	StartupPressureBaseValue	:	REAL;

	ton_StartupRetryTimer		: 	TON := (PT := T#10S);
	Ton_StartupFailedTimer		:	TON := (PT := T#1M);
	TP_PumpRetryDelay			:	Tp := (Pt := T#2S);
	
	rTrig_PumpStarted			:	r_Trig;
	
	b_test		:	BOOL;
END_VAR
Tp_PumpRetryDelay(IN := ton_StartupRetryTimer.Q);
ton_StartupRetryTimer(IN:= Outputs.DCPumpEnable);
Ton_StartupFailedTimer(IN:= DCPumpState = ePumpState.Starting);


rTrig_PumpStarted(clk := outputs.DCPumpEnable);
IF rTrig_PumpStarted.Q THEN
	StartupPressureBaseValue := r_CoolantPressure;
END_IF

CASE DCPumpState OF
	ePumpState.Off:
		outputs.DCPumpEnable := FALSE;
		IF b_24VDCavailable THEN
			DCPumpState := ePumpState.Starting;
			Events.b_DCpumpTimeout := FALSE;
		END_IF
		
	ePumpState.Starting:
		//enable pump power unless waiting for a retry
		outputs.DCPumpEnable := NOT TP_PumpRetryDelay.Q;
		
		IF TP_PumpRetryDelay.Q THEN
			Events.b_DCpumpTimeout := TRUE;
		END_IF
			
		//Switch to running mode if presure rise is reached
		IF (r_CoolantPressure - StartupPressureBaseValue) > st_params.r_StartupPumpMinimumPressure THEN
			DCPumpState := ePumpState.Running;
			Events.b_DCpumpTimeout := FALSE;
		END_IF
		
		//if startup takes too long. stop trying and raise event.	
		IF Ton_StartupFailedTimer.Q THEN
	Events.b_DCpumpPressureFault := TRUE;
			DCPumpState := ePumpState.Off;
		END_IF
	
	ePumpState.Running:
		outputs.DCPumpEnable := TRUE;
		IF NOT b_24VDCAvailable THEN
			DCPumpState := ePumpState.OFF;
END_IF

	ePumpState.Stopping:
		outputs.DCPumpEnable := FALSE;
		DCPumpState := ePumpState.OFF;
end_case

		
DCPumpOn	:=	DCPumpState = ePumpState.Running;
END_METHOD

METHOD PRIVATE DisableBatteryLoop : BOOL
VAR_INPUT
END_VAR
Outputs.BattLoopValveClose := TRUE;
DisableBatteryLoop := NOT inputs.BattLoopValveFB;
END_METHOD

METHOD PRIVATE DisableFanCoilLoop : BOOL
VAR_INPUT
END_VAR
Outputs.FancoilLoopValveClose := TRUE;
DisableFancoilLoop := NOT inputs.FancoilLoopValveFB;
END_METHOD

METHOD PRIVATE DisableInverterLoop : BOOL
VAR_INPUT
END_VAR
IF NOT b_inverterrunning THEN
	Outputs.InvLoopValveClose := TRUE;
ELSE
	Outputs.InvLoopValveClose := FALSE;
END_IF

DisableInverterLoop := NOT inputs.InvloopValveFB;
END_METHOD

METHOD EnclosureCooling : BOOL
VAR_INPUT
END_VAR
outputs.DCFanEnable	:= TRUE;
EnclosureCooling := DisableInverterLoop() AND DCPumpOn();
END_METHOD

METHOD FullCooling : BOOL
VAR_INPUT
END_VAR

VAR_INST
	Pumpfb : BOOL;
END_VAR
Outputs.InvLoopValveClose := FALSE;

IF ACPumpON() THEN
	PumpFb := TRUE;
	DCPumpOFF(FALSE);
	Outputs.FancoilLoopValveClose := FALSE;
	Outputs.BattLoopValveClose := FALSE;
ELSE
	PumpFb := FALSE;
	Outputs.FancoilLoopValveClose := TRUE;
	Outputs.BattLoopValveClose := TRUE;
	DCpumpON();
END_IF



FullCooling := 
	inputs.BattLoopValveFB 
	//AND inputs.FancoilLoopValveFB 
	AND inputs.InvLoopValveFB
	AND PumpFb;
END_METHOD

METHOD PRIVATE GetCoolantData : BOOL

VAR_INPUT
	Pwarning		: REAL;
	PError			: REAL;
	PHyst			: REAL;
END_VAR


VAR_INST
	Ton_IdlePressureDelayTimer	:	TON := (PT:= T#1m);
	SR_IdlePressureWarning		: SR;
	SR_IdlePressureError		: SR;
END_VAR
r_CoolantPressure := (INT_TO_REAL(Inputs.CoolingLoopPressureSensor)/16#7FFF * 4);
r_CoolantTemperature := INT_TO_REAL(Inputs.CoolingLoopTemperatureSensor) / 10 ;

Ton_IdlePressureDelayTimer(in:= NOT (outputs.ACPumpEnable OR Outputs.DCPumpEnable));
IF ton_idlePressureDelayTimer.Q THEN
	r_CoolantidlePressure := r_CoolantPressure;
END_IF

// generate events
SR_Idlepressurewarning(set1:=  (r_CoolantPressure < Pwarning),
						RESET:=  (r_CoolantPressure > (Pwarning + PHyst)),
						Q1 => events.b_CoolingLoopIdlePressureWarning);
SR_IdlepressureError(set1:=  (r_CoolantPressure < Perror),
						RESET:=  (r_CoolantPressure > (Perror + PHyst)),
						Q1 => events.b_CoolingLoopIdlePressureError);
END_METHOD

METHOD GetWearCounters : BOOL
VAR_INST
	ACPumpCycles			:	FB_Varlogger;
	ACPumpHours				:	FB_Varlogger;
	DCPumpCycles			:	FB_Varlogger;
	DCPumpHours				:	FB_Varlogger;
	
	BattValveCycles			:	FB_Varlogger;
	InverterValveCycles		:	FB_Varlogger;
	FancoilValveCycles		:	FB_Varlogger;
	
	DCFanCycles				:	FB_Varlogger;
	DCFanHours				:	FB_Varlogger;
	

		
	
	PrechargeCycleLogger	:	FB_Varlogger;
	SOHLogger				:	FB_Varlogger;
	CycleCountLogger		:	FB_Varlogger;
	OvertempCountLogger		:	FB_Varlogger;
	OverTempTimeLogger		:	FB_Varlogger;
	UnderTempCountLogger	:	FB_Varlogger;
	UnderTempTimeLogger		:	FB_Varlogger;
	EnergyInLogger			:	FB_Varlogger;
	EnergyOutLogger			:	FB_Varlogger;
END_VAR

ACPumpCycles(			TriggerInput := Outputs.ACPumpEnable,
						LogItemGroup := eLogItemGroupID.CoolingSystem, 
						LogItemName := 'ACPumpCnt', 
						LogType := eLogTypes.TrackCycles);

ACPumpHours(			TriggerInput := Outputs.ACPumpEnable,
						LogItemGroup := eLogItemGroupID.CoolingSystem, 
						LogItemName := 'ACPumpHrs', 
						LogType := eLogTypes.TrackOnTime);
						
DCPumpCycles(			TriggerInput := Outputs.DCPumpEnable, 
						LogItemGroup :=  eLogItemGroupID.CoolingSystem, 
						LogItemName := 'DCPumpCnt', 
						LogType := eLogTypes.TrackCycles);	

DCPumpHours(			TriggerInput := Outputs.DCPumpEnable, 
						LogItemGroup :=  eLogItemGroupID.CoolingSystem, 
						LogItemName := 'DCPumpHrs', 
						LogType := eLogTypes.TrackOnTime);	

BattValveCycles(		TriggerInput := outputs.BattLoopValveClose, 
						LogItemGroup :=  eLogItemGroupID.CoolingSystem, 
						LogItemName := 'BattValveCnt', 
						LogType := eLogTypes.TrackCycles);		
						
InverterValveCycles(	TriggerInput := outputs.InvLoopValveClose, 
						LogItemGroup :=  eLogItemGroupID.CoolingSystem, 
						LogItemName := 'InvValveCnt', 
						LogType := eLogTypes.TrackCycles);	
						
FancoilValveCycles(		TriggerInput := outputs.FancoilLoopValveClose, 
						LogItemGroup :=  eLogItemGroupID.CoolingSystem, 
						LogItemName := 'FancoilValveCnt', 
						LogType := eLogTypes.TrackCycles);	
												
DCFanCycles(			TriggerInput := Outputs.DCFanEnable, 
						LogItemGroup :=  eLogItemGroupID.CoolingSystem, 
						LogItemName := 'DCFanCnt', 
						LogType := eLogTypes.TrackCycles);	

DCFanHours(				TriggerInput := Outputs.DCFanEnable, 
						LogItemGroup :=  eLogItemGroupID.CoolingSystem, 
						LogItemName := 'DCFanHrs', 
						LogType := eLogTypes.TrackOnTime);
END_METHOD

METHOD Idle : BOOL
VAR_INPUT
	force	: BOOL;
END_VAR

VAR_INST
	PumpFbOff		: BOOL;
END_VAR
outputs.DCFanEnable	:= FALSE;

IF NOT b_inverterRunning THEN
	PumpFBOff := DCPumpOff(force) AND ACpumpOff();
	Outputs.FancoilLoopValveClose := FALSE;
	Outputs.BattLoopValveClose := FALSE;
	Outputs.InvLoopValveClose := FALSE;
ELSE
	Outputs.FancoilLoopValveClose := TRUE;
	Outputs.BattLoopValveClose := TRUE;
	PumpFbOff := NOT DCPumpOn();
END_IF

Idle := PumpFBOff;
END_METHOD

METHOD LimitedCooling : BOOL

VAR_INST
	pumpfb	: BOOL;
	fb		: BOOL;
END_VAR
Outputs.FancoilLoopValveClose := TRUE;
Outputs.BattLoopValveClose :=  TRUE;
Outputs.InvLoopValveClose := FALSE;


IF DCPumpON() THEN
	pumpfb := ACPumpOFF();
ELSE
	pumpfb := FALSE;
END_IF

//feedback
fb := 
	NOT inputs.BattLoopValveFB 
	AND NOT inputs.FancoilLoopValveFB 
	AND inputs.InvLoopValveFB 
	AND pumpfb;
	
LimitedCooling := fb;
END_METHOD

END_FUNCTION_BLOCK

// ---- POUs/Objects/PowerStack/FB_PowerStack.TcPOU
FUNCTION_BLOCK FB_PowerStack
//Accessible input data from main program
VAR_INPUT
	set											: ST_PowerStack_Set;
	e_ACRotationStateExt						: eACRotationState;
	b_EnableFan									: BOOL;
	b_transportMode								: BOOL;
	b_rotationswitchEnable						: BOOL;
	by_CoolingPowerRequest						: BYTE; //0 off, 1 internal 400VAC supply required, 2 Full Power Allowed
	r_PLossInternal								: REAL;
	r_QLossInternal								: REAL;
	b_DoublePowermodule							: BOOL;	
	b_BatteryDCReady							: BOOL;	
	r_BatteryDCVoltage							: REAL;
	b_ExtGridCodeTrip							: BOOL;	
	b_OutputConnected							: BOOL;
	b_InputConnected							: BOOL;
	b_InternalACRequired						: BOOL;
END_VAR

//Accessible output data to main program
VAR_OUTPUT
	get										: ST_PowerStack_Get;
	st_InternalPsuSupplyRequest				: ST_InternalPowerSupply_PowerDemand;
	b_InternalPsuACOk						: BOOL;
	b_MasterMccbEDM							: BOOL;
	b_SlaveMccbEDM							: BOOL;
	b_NetcontEDM							: BOOL;
	by_CoolingControl						: BYTE; // 0:= off, 1:= startup, 2:= run
END_VAR

//These variables MUST be passed to the powerstack in order to work properly. Thats why they are declared separately in the VAR_IN_OUT (CONSTANT)
VAR_IN_OUT CONSTANT			
	st_params									: ST_Powerstack_Params;
	st_calibration								: ST_Powerstack_calibration;
END_VAR

// local variables in powerstack
VAR
	//function blocks
	Netcontactor						: FB_Netcontactor;
	PowermoduleMaster					: FB_powermodule;
	PowermoduleSlave					: FB_powermodule;
	LOM 								: FB_LOMDetection;
END_VAR

VAR
    eControl 					: (stand_by, Start, Stop, Shutdown);
	s_ErrorStep					: STRING;
	rTrig_start					: R_Trig;
	ton_StandbyNetConCloseDelay : TON := (PT:= T#5S);
	ton_SFCtipDelay				: TON := (PT:= T#1S);
	
	standbyDeactivateState		: BOOL; // trigger on shutdown, reset on busbar ac Rtrig or Reset.
	rTrig_StandByDeactStateReset: R_TRIG;
END_VAR

Netcontactor();
	get.Netcontactor REF= netcontactor.get;
	Netcontactor.set.e_ACRotationState := e_ACRotationStateExt;
	Netcontactor.set.b_ACdetected := get.b_ACDetected;
	Netcontactor.set.b_RotationSwitchEnable := b_rotationswitchEnable;
	Netcontactor.set.e_ClosingRequest := set.e_NetconClosingRequest;
	Netcontactor.set.b_SynchronizedToD7	:= PowermoduleMaster.get.UgridStatusWord.b_SynchronizedToD7;
	PowermoduleMaster.set.b_D7SyncRequest := Netcontactor.get.b_SyncCloseCommand;
	

 //passthrough the reference of the get/set input and output variables to underlaying functions.
PowermoduleMaster(
	b_enable := TRUE,
	 st_params:=st_params.PowermoduleMaster,
	st_calibration := st_calibration.Master,
	e_ID := eObject_ID.PowerModuleMaster,
	r_batteryDCVoltage := r_BatteryDCVoltage);
	get.PowermoduleMaster REF= powermoduleMaster.get;
PowermoduleSlave(
	b_enable := b_doublePowermodule,
 	st_params:=st_params.PowermoduleSlave, 
	st_calibration := st_calibration.Slave,
	e_ID := eObject_ID.PowerModuleSlave,
	r_batteryDCVoltage := r_BatteryDCVoltage);
	get.PowermoduleSlave REF= powermoduleSlave.get;
	
//Start Stop sequence
StartStopSFC();

//Bundle data from powermodules to powerstack total
BundlePowerStackGets(st_params := st_params);

//Droop settings to/from powermodules
ControlDroop(
	setMaster := powermoduleMaster.set,
	setSlave := powerModuleSlave.set,
	b_ControlEnabled := get.b_ControlEnabled
	);

//Powermodules Control
Controlpowermodules(
	r_APloss:= r_PLossInternal,
	r_RPloss := r_QLossInternal,
	setMaster:= Powermodulemaster.set,
	setSlave:= PowermoduleSlave.set,
	st_params := st_params);

//setEvents
setEvents(events:= get.Events,  st_params := St_params);

b_MasterMccbEDM	:= PowermoduleMaster.b_MccbEDM;
b_SlaveMccbEDM	:= PowermoduleSlave.b_MccbEDM;
b_NetContEDM	:= Netcontactor.b_NetcontEDM;

//start trigger
rTrig_start(CLK:= eControl = Start);

ACTION _aCloseNetcontactor_active:
get.e_State 				:= eStatusPowerStack.synchronization;

IF (NOT ton_StandbyNetConCloseDelay.Q OR standbyDeactivateState) AND eControl = stand_by THEN
	SFCtip := NOT SFCTIP;
ELSE
	SFCtip := Netcontactor.Close(b_Force := NOT get.b_ACDetected) AND NOT SFCTIP;
END_IF
END_ACTION

ACTION _aContinousActions:
IF SFCerror THEN s_ErrorStep := SFCCurrentStep; END_IF;

//evaluate if inverter is in a gridforming kinda mode
get.b_InverterGridFormingMode := get.e_InverterMode <> eInvertermodes.Afe AND get.e_PowerMode <> ePowermodes.Isochronous AND get.b_InverterRunning;

//busbar AC check	
get.b_ACDetected := AcCheck(get.r_ACVoltageD7, get.r_FrequencyD7);

// evaluate grid AC, or when grid is lost.
DetectGridSync(
	b_netconFB := netcontactor.get.b_NetConFb,
	b_InverterGridFormingMode := get.b_InverterGridFormingMode,
	b_ExtGridConnected := set.b_ExtGridConnected,
	b_ACOk := get.b_ACDetected,
	b_IsochroneMode := powermodulemaster.get.e_PowerMode = ePowermodes.Isochronous,
	b_gridtied := get.b_GridTied,
	b_ACdetected := get.b_GridACdetected,
	b_GridCodeTripInverter := Powermodulemaster.get.GridcodeStatusWord.b_GridCodeTripActive,
	b_GridCodeActiveInverter := powermodulemaster.get.controldata.Controlword.b_GridCodeEnable,
	b_GridCodeOK := get.b_GridCodeOK,
	b_GridCheckActive := get.b_GridCodeCheckActive,
	t_GridLostMaxTripTime := TO_TIME(Settings.GridParams.ui_GCTripMaxTripTime),
	t_GridOKReleaseTime :=  TO_TIME(TO_REAL(settings.GridParams.ui_GCokReleaseTime)*1000)
	);



//Evaluate ac available for standby mode
ton_StandbyNetConCloseDelay(IN := st_params.b_StandbyEnable 
	AND get.b_GridACdetected
	AND set.b_automaticswitching);	
	
// internal AC check
//b_InternalPsuACOk := InternalAcCheck(SEL(netcontactor.get.b_NetConFb, get.r_ACVoltageSupply, get.r_ACVoltageD7), get.r_FrequencySupply, get.b_GridTied);
b_InternalPsuACOk := InternalAcCheck(	SEL(netcontactor.get.b_NetConFb, get.r_ACVoltageSupply, get.r_ACVoltageD7), 
										SEL(netcontactor.get.b_NetConFb, get.r_FrequencySupply, get.r_FrequencyD7));


//get starting enable condition
get.b_StartEnabled := StartingEnable();

rTrig_StandByDeactStateReset(CLK:= get.b_ACDetected);
IF rTrig_standbyDeactStateReset.Q THEN
	standbyDeactivateState := FALSE;
END_IF
END_ACTION

ACTION _aCoolingRequest_active:
by_CoolingControl := 1;

get.e_State := eStatusPowerStack.Wait_CoolingMode1;
END_ACTION

ACTION _aHVDCRequest_active:
st_InternalPsuSupplyRequest.b_Demand_HVDC := TRUE;
get.e_State := eStatusPowerStack.Wait_HVDC;
END_ACTION

ACTION _aIdle_active:
get.events.b_GridCodeWarning:= FALSE; 
get.b_ControlEnabled		:= TRUE;


IF Netcontactor.Open() AND PowermoduleMaster.Idle() THEN
	get.b_StartedState 			:= FALSE;
	get.e_State := eStatusPowerStack.idle;
	//PowermoduleMaster.Idle();
	IF get.b_GridCodeOK THEN
		get.e_State 							:= eStatusPowerStack.GridCodeStop;
	END_IF
END_IF



//SFCtip := XNOR((get.b_GridCodeOK AND get.b_GridCodeCheckActive), eControl = start) AND NOT detectConnectionLoss(TRUE) AND NOT SFCtip;
SFCtip := SEL(get.b_GridCodeCheckActive, TRUE, get.b_GridCodeOK) AND eControl = start AND NOT detectConnectionLoss(TRUE) AND NOT SFCtip;
//IF get.b_GridACdetected AND get.Netcontactor.b_NetConFb THEN
//	PowermoduleMaster.Idle(); //Stop modulation to stop power supply when grid is existing. Grid supplies internals through net contactor
//ELSE
//	Netcontactor.Open(); // keep master inverter modulation, but open netcontactor to stop power supply to load.
//END_IF

//PowermoduleSlave.Idle(); //stop slave always
END_ACTION

ACTION _aInit_active:
SFCReset 					:= FALSE;
get.b_StartedState 			:= FALSE;

get.e_State := eStatusPowerStack.Init;
get.b_ControlEnabled 	:= FALSE;

//IF by_CoolingPowerRequest = eCoolingPowerRequest.off THEN
IF NOT b_internalACRequired THEN
	ShutdownFull(FALSE);
	IF NOT get.b_ACDetected THEN
		Netcontactor.Open();
	END_IF
ELSE
	get.e_State := eStatusPowerstack.Cooling_Shutdown;
END_IF

//by_CoolingControl		:= 0;
//b_InternalPsuACOk		:= FALSE;
END_ACTION

ACTION _aRunning_active:
get.b_ControlEnabled		:= TRUE;
get.b_StartedState 			:= TRUE;
PowermoduleMaster.Run(set.e_PowerMode, set.e_InverterMode, NOT netcontactor.get.b_NetConFb);
get.e_State 				:= eStatusPowerStack.running;

//If force close is activated, the gridcode trip will be not lead to opening of the contactor.
//this is used to operate an external contactor instead.
IF set.b_NetcontactorHoldClose AND netcontactor.get.b_NetConFb THEN
	Netcontactor.Close(TRUE);
	SFCTip := DetectConnectionLoss(FALSE) AND NOT SFCTip;
ELSE 
	SFCtip := LOM.Q OR (NOT get.b_GridCodeOK AND get.b_GridCodeCheckActive) OR DetectConnectionLoss(TRUE) OR by_CoolingPowerRequest <> 2 AND NOT SFCTip;
END_IF
END_ACTION

ACTION _aSFCtip_reset:
sfctip:= FALSE;
END_ACTION

ACTION _aStandBy_active:
//default values, will be overwritten if neccessary
get.e_State := eStatusPowerstack.Standby;
PowermoduleSlave.Shutdown(b_force := FALSE);// slave shutdown always during stand-by

IF get.b_InverterRunning THEN
	by_CoolingControl := 1;
ELSE 
	by_CoolingControl := 0;	// Also cooling deactivated from a powermodule point of view. Cooling decides if this can be achieved.
END_IF

	
ton_SFCtipDelay(Q=> SFCtip);

IF st_params.b_StandbyEnable AND set.b_automaticswitching AND NOT b_transportMode AND b_InternalACRequired THEN
	IF ton_StandbyNetconCloseDelay.Q THEN // if grid, than close netcontactor
		get.e_State := eStatusPowerstack.Standby_GridSupply;	
		IF NOT Netcontactor.get.b_NetConFb AND NOT st_params.b_SoftStartEnable AND NOT get.b_InverterRunning THEN
			Netcontactor.Close(TRUE);
		//ELSIF NOT Netcontactor.get.b_NetConFb AND NOT standbyDeactivateState THEN
			//ton_SFCtipDelay.IN:= NOT ton_SFCtipDelay.Q;
		//ELSIF by_CoolingPowerRequest = eCoolingPowerRequest.off THEN
		ELSIF NOT b_InternalACRequired THEN
			ShutdownFull(FALSE);
		ELSIF get.b_InverterRunning AND Netcontactor.get.b_NetConFb THEN
			PowermoduleMaster.Run(ePowermodes.Isochronous ,eInverterModes.Microgrid, FALSE);
		ELSIF (b_InternalACRequired AND NOT standbyDeactivateState AND (NOT get.b_InverterRunning OR NOT Netcontactor.get.b_NetConFb)) THEN
			ton_SFCtipDelay.IN:= NOT ton_SFCtipDelay.Q;
		END_IF
	//if no grid detected, no internal supply is made by default unless it is requested from cooling	
	ELSIF Netcontactor.Open() THEN
		//IF by_CoolingPowerRequest = eCoolingPowerRequest.off THEN
		IF NOT b_InternalACRequired THEN
			ShutdownFull(FALSE);	
		ELSE
			ton_SFCtipDelay.IN:= NOT ton_SFCtipDelay.Q AND NOT PowermoduleMaster.Run(ePowermodes.Droop, eInverterModes.Island, TRUE);
		END_IF
		get.e_State := eStatusPowerstack.Standby_InternalSupply;
	END_IF
ELSE
	IF NOT get.b_GridACdetected THEN
		Netcontactor.Open();
	END_IF
	
	//IF by_CoolingPowerRequest = eCoolingPowerRequest.off THEN
	IF NOT b_InternalACRequired THEN
		IF Netcontactor.Open() AND ShutdownFull(FALSE) THEN
			get.e_State := eStatusPowerstack.Standby;
		END_IF
	ELSE
		get.e_State := eStatusPowerstack.Cooling_Shutdown;
	END_IF
END_IF
END_ACTION

ACTION _aStandby_exit:
SFCtip := FALSE;
ton_SFCtipDelay.IN := FALSE;

IF eControl = start THEN 
	ton_StandbyNetConCloseDelay.IN := FALSE;
END_IF

st_InternalPsuSupplyRequest.b_Demand_24V := TRUE;
END_ACTION

ACTION _aStartMaster_active:
sfctip := PowermoduleMaster.Start(netcontactor.get.b_NetConFb AND get.b_ACdetected) AND NOT SFCTip;
get.e_State := eStatusPowerStack.Start_Master;
END_ACTION

ACTION _aStartSlave_active:
sfctip:= PowermoduleSlave.Start(TRUE);
get.e_State 		:= eStatusPowerStack.Start_Slave;
END_ACTION

ACTION _aUVRSupplyRequest_active:
IF b_doublePowermodule THEN
	SFCtip := powermodulemaster.get.b_MccbUvr24VdcOK AND powermoduleSlave.get.b_MccbUvr24VdcOK AND NOT SFCtip;
ELSE
	SFCtip := powermodulemaster.get.b_MccbUvr24VdcOK AND NOT SFCtip;
END_IF
END_ACTION

METHOD PRIVATE BundlePowerStackGets : BOOL
VAR_IN_OUT CONSTANT
	st_params			: ST_Powerstack_params;
END_VAR
VAR_INST
	r_Derating : REAL;
END_VAR
get.e_PowerMode			:= get.PowermoduleMaster.e_PowerMode;
get.r_FrequencySupply := get.PowermoduleMaster.r_FrequencySupply;
get.r_ACVoltageSupply	:= get.PowermoduleMaster.r_ACVoltageSupply;
get.r_ACVoltageD7		:= get.PowermoduleMaster.r_ACVoltageD7;
get.r_FrequencyD7		:= get.PowermoduleMaster.r_FrequencyD7;
get.r_FrequencyDroop	:= get.PowermoduleMaster.r_FrequencyDroop;
get.r_VoltageDroop		:= get.PowermoduleMaster.r_VoltageDroop;

get.r_ActivePower		:= get.PowermoduleMaster.r_ActivePower + get.PowermoduleSlave.r_ActivePower;
get.r_ReactivePower		:= get.PowermoduleMaster.r_ReactivePower + get.PowermoduleSlave.r_ReactivePower;
get.r_ApparentPower		:= get.PowermoduleMaster.r_ApparentPower + get.PowermoduleSlave.r_ApparentPower;
get.r_CosPhi			:= SEL(get.r_ApparentPower = 0, (get.r_ActivePower / get.r_ApparentPower), 0); //avoid dividing by zero;
get.r_DCcurrent			:= get.PowermoduleMaster.r_DCCurrent	+ get.PowermoduleSlave.r_DCCurrent;
get.r_DCVoltage			:= get.PowermoduleMaster.r_DCVoltage;
get.r_DCPower			:= get.PowermoduleMaster.r_DCPower + get.PowermoduleSlave.r_DCPower;
get.r_LoadPercent		:= SEL(
	b_DoublePowermodule,get.PowermoduleMaster.r_LoadPercent, (get.PowermoduleMaster.r_LoadPercent + get.PowermoduleSlave.r_LoadPercent) / 2);
get.r_Pmin				:= get.PowermoduleMaster.r_Pmin + get.PowermoduleSlave.r_Pmin;
get.r_Pmax				:= get.PowermoduleMaster.r_Pmax + get.PowermoduleSlave.r_Pmax;
get.r_QMax				:= get.PowermoduleMaster.r_Qmax + get.PowermoduleSlave.r_Qmax;
get.r_QMin				:= get.PowermoduleMaster.r_Qmin + get.PowermoduleSlave.r_Qmin;
get.r_ACcurrentLimit	:= get.PowermoduleMaster.r_ACcurrentLimit + get.PowermoduleSlave.r_ACcurrentLimit;
get.r_ACcurrentLimitMax	:= SEL(b_doublePowermodule, st_params.PowermoduleMaster.r_ACCurrentLimitMax, st_params.PowermoduleMaster.r_ACCurrentLimitMax + st_params.PowermoduleSlave.r_ACCurrentLimitMax);
get.r_Smax				:= get.r_ACcurrentLimit * get.r_ACVoltageSupply * 1.73 / 1000; 
get.r_PowerChangeRate	:= TO_REAL(st_params.i_MaxPowerChangeRate);
get.r_AcCurrent	:= get.PowermoduleMaster.r_ACCurrent + get.PowermoduleSlave.r_ACCurrent;


get.r_OvercurrentValueAct 	:= SEL(
	b_DoublePowermodule, 
	get.PowermoduleMaster.r_OverCurrentValue, 
	(get.PowermoduleMaster.r_OverCurrentValue + get.PowermoduleSlave.r_OverCurrentValue) / 2
	);
get.r_ThrottlingValueAct := (1 - LIMIT(0, get.r_OvercurrentValueAct, 1)) * 100;
	
get.b_inverterRunning 	:= PowermoduleMaster.get.StatusWord.b_Running OR PowermoduleSlave.get.StatusWord.b_Running;
get.b_DCDetected 		:= powermoduleMaster.get.r_DCVoltage > 120; // vdc
get.r_OvercurrentValueMax:= TO_REAL(st_params.ui_OvercurrentRating) /100;
r_Derating := (100 - TO_REAL(st_params.ui_DeratingStack)) / 100; // total current derating when parallel inverters according to danfoss
get.r_RatedCurrent 	:= (st_params.powermodulemaster.r_InverterRatedCurrent + SEL(b_doublePowermodule,0,st_params.PowermoduleSlave.r_InverterRatedCurrent * r_Derating));
get.r_RatedPower	:= (st_params.powermodulemaster.r_InverterRatedPower + SEL(b_doublePowermodule,0,st_params.PowermoduleSlave.r_InverterRatedPower* r_Derating));

get.b_EcomodeAvailable := b_DoublePowermodule;

get.r_MaxTemperature := MAX(powermodulemaster.get.r_TemperatureMax, powermoduleSlave.get.r_TemperatureMax);
//get.b_GridCodeOK := NOT powermodulemaster.get.GridcodeStatusWord.b_GridCodeTripActive;
//get.b_GridCodeActive := powermodulemaster.get.controldata.Controlword.b_GridCodeEnable;
get.e_InverterMode := powermodulemaster.get.e_InverterMode;
get.e_PowerMode := powermodulemaster.get.e_PowerMode;
get.e_ThrottlingStatus := powermodulemaster.get.e_ThrottlingStatus;

IF get.r_ActivePower > 1 THEN
	get.e_PowerState := ePowerstate.Discharging;
ELSIF get.r_ActivePower < 1 THEN
	get.e_PowerState := ePowerstate.Charging;
ELSE
	get.e_PowerState := ePowerstate.None;
END_IF
END_METHOD

METHOD PRIVATE ControlDroop
VAR_IN_OUT
	setMaster			: ST_Powermodule_Set;
	setSlave			: ST_Powermodule_Set;
	b_controlEnabled	: BOOL;
END_VAR

VAR
	r_DroopLimitMin		: REAL;
	r_DroopLimitMax		: REAL;
END_VAR
r_DroopLimitMin := LIMIT(0,st_params.r_DroopMinimum, st_params.r_DroopMaximum );
r_DroopLimitMax := MAX(st_params.r_DroopMinimum, st_params.r_DroopMaximum);

//Write to powermodules
setMaster.r_FrequencyDroop	:= LIMIT(r_DroopLimitMin, set.r_FrequencyDroop, r_DroopLimitMax);
setMaster.r_VoltageDroop	:= LIMIT(r_DroopLimitMin, set.r_VoltageDroop,	r_DroopLimitMax);
setSlave.r_FrequencyDroop	:= LIMIT(r_DroopLimitMin, set.r_FrequencyDroop,	r_DroopLimitMax);
setSlave.r_VoltageDroop 	:= LIMIT(r_DroopLimitMin, set.r_VoltageDroop,	r_DroopLimitMax); 


// read from powermodules
IF NOT b_ControlEnabled THEN				//during startup control is disabled and the powermode only from first inverter. 
	get.e_PowerMode := get.PowermoduleMaster.e_PowerMode;
ELSE
	IF get.PowermoduleMaster.e_PowerMode = ePowerModes.Droop AND SEL(Settings.Configuration.b_DoublePowerModule, 1, get.PowermoduleSlave.e_PowerMode = ePowerModes.Droop) THEN
		get.e_PowerMode:= ePowerModes.Droop;
	ELSIF get.PowermoduleMaster.e_PowerMode = ePowerModes.DroopZeroStart AND SEL(Settings.Configuration.b_DoublePowerModule, 1, get.PowermoduleSlave.e_PowerMode = ePowerModes.DroopZeroStart) THEN
		get.e_PowerMode := ePowerModes.DroopZeroStart;
	ELSIF get.PowermoduleMaster.e_PowerMode = ePowerModes.Isochronous AND SEL(Settings.Configuration.b_DoublePowerModule, 1, get.PowermoduleSlave.e_PowerMode = ePowerModes.Isochronous) THEN
		get.e_PowerMode := ePowerModes.Isochronous;
	END_IF
END_IF
END_METHOD

METHOD PRIVATE ControlPowermodules : BOOL

VAR_IN_OUT CONSTANT
	r_APloss	: REAL;
	r_RPloss	: REAL;
	st_params 	: ST_Powerstack_params;
END_VAR

VAR_IN_OUT
	setMaster			: ST_Powermodule_Set;
	setSlave			: ST_Powermodule_Set;
END_VAR

VAR_INST
	r_PmaxFinal						: REAL;
	r_PminFinal						: REAL;
	r_PLMfreqOffset					: REAL;
	r_PLMvoltOffset					: REAL;
	r_FreqDeltaLOM					: REAL;	
	ton_GridCodeTripDelay			: TON := (PT:= T#2S);
	ton_RampDisabled				: Ton := (PT := T#2S);
	fb_ramp_Pset					: fb_Ramp := (b_Enable := TRUE, r_rampRate := 50);
	fb_ramp_Qset					: fb_Ramp := (b_Enable := TRUE, r_rampRate := 50);
	r_Derating						: REAL;
	r_PM1Load						: REAL; // 0- 100 %
	r_PM2Load						: REAL; // 0- 100 % 
	r_GrossActivePower				: REAL;
	r_GrossReactivePower			: REAL;
	r_ActiveLossOffset				: REAL;
	r_ReactiveLossOffset			: REAL;
	
	// Nominal Voltage and frequency
	r_VoltageDroopOffset				: REAL;
	r_FrequencyDroopOffset				: REAL;
	
	r_Pmax			: REAL;
	r_Pmin			: REAL;
	r_ACcurrentLimit: REAL;
END_VAR
// Variables to be used in the controls
r_PM1Load := SEL(b_doublePowermodule, 1, st_params.PowermoduleMaster.r_InverterRatedCurrent / get.r_RatedCurrent);
r_PM2Load := 1- r_PM1Load; // Same as 1- r_contributionPM1


//write to powermodules
//set island mode
setMaster.r_DroopIslandMode := st_params.r_DroopIslandMode;
setMaster.r_DroopMaximum := st_params.r_DroopMaximum;
setMaster.r_DroopMinimum := st_params.r_DroopMinimum;

//Control fan
setMaster.b_FanContactor := b_EnableFan;
setSlave.b_FanContactor := b_EnableFan;

